LIN {X 0,Y 573.256,Z 464.198,A -85,B 0,C 180,E1 -2012.645,E2 -2012.645} C_VEL
LIN {X 0,Y 573.257,Z 464.201,A -85,B 0,C 180,E1 -2015.184,E2 -2015.184} C_VEL
LIN {X 0,Y 573.236,Z 464.206,A -85,B 0,C 180,E1 -2017.808,E2 -2017.808} C_VEL
LIN {X 0,Y 573.247,Z 464.198,A -85,B 0,C 180,E1 -2020.525,E2 -2020.525} C_VEL
LIN {X 0,Y 573.239,Z 464.205,A -85,B 0,C 180,E1 -2023.359,E2 -2023.359} C_VEL
LIN {X 0,Y 573.256,Z 464.197,A -85,B 0,C 180,E1 -2026.33,E2 -2026.33} C_VEL
LIN {X 0,Y 573.242,Z 464.198,A -85,B 0,C 180,E1 -2028.544,E2 -2028.544} C_VEL
LIN {X 0,Y 573.245,Z 464.204,A -85,B 0,C 180,E1 -2031.298,E2 -2031.298} C_VEL
LIN {X 0,Y 573.215,Z 464.205,A -85,B 0,C 180,E1 -2034.018,E2 -2034.018} C_VEL
LIN {X 0,Y 573.272,Z 464.195,A -85,B 0,C 180,E1 -2036.518,E2 -2036.518} C_VEL
LIN {X 0,Y 573.232,Z 464.203,A -85,B 0,C 180,E1 -2039.118,E2 -2039.118} C_VEL
LIN {X 0,Y 573.255,Z 464.2,A -85,B 0,C 180,E1 -2041.971,E2 -2041.971} C_VEL
LIN {X 0,Y 573.255,Z 464.197,A -85,B 0,C 180,E1 -2044.59,E2 -2044.59} C_VEL
LIN {X 0,Y 573.238,Z 464.207,A -85,B 0,C 180,E1 -2047.662,E2 -2047.662} C_VEL
LIN {X 0,Y 573.278,Z 464.194,A -85,B 0,C 180,E1 -2050.67,E2 -2050.67} C_VEL
LIN {X 0,Y 573.256,Z 464.205,A -85,B 0,C 180,E1 -2053.622,E2 -2053.622} C_VEL
LIN {X 0,Y 573.276,Z 464.199,A -85,B 0,C 180,E1 -2055.807,E2 -2055.807} C_VEL
LIN {X 0,Y 573.265,Z 464.196,A -85,B 0,C 180,E1 -2058.745,E2 -2058.745} C_VEL
LIN {X 0,Y 573.309,Z 464.199,A -85,B 0,C 180,E1 -2061.541,E2 -2061.541} C_VEL
LIN {X 0,Y 573.291,Z 464.192,A -85,B 0,C 180,E1 -2064.372,E2 -2064.372} C_VEL
LIN {X 0,Y 573.316,Z 464.193,A -85,B 0,C 180,E1 -2067.892,E2 -2067.892} C_VEL
LIN {X 0,Y 573.33,Z 464.188,A -85,B 0,C 180,E1 -2070.702,E2 -2070.702} C_VEL
LIN {X 0,Y 573.306,Z 464.192,A -85,B 0,C 180,E1 -2072.811,E2 -2072.811} C_VEL
LIN {X 0,Y 573.301,Z 464.198,A -85,B 0,C 180,E1 -2075.628,E2 -2075.628} C_VEL
LIN {X 0,Y 573.286,Z 464.193,A -85,B 0,C 180,E1 -2078.459,E2 -2078.459} C_VEL
LIN {X 0,Y 573.274,Z 464.203,A -85,B 0,C 180,E1 -2081.312,E2 -2081.312} C_VEL
LIN {X 0,Y 573.284,Z 464.193,A -85,B 0,C 180,E1 -2084.425,E2 -2084.425} C_VEL
LIN {X 0,Y 573.261,Z 464.202,A -85,B 0,C 180,E1 -2087.112,E2 -2087.112} C_VEL
LIN {X 0,Y 573.254,Z 464.198,A -85,B 0,C 180,E1 -2090.077,E2 -2090.077} C_VEL
LIN {X 0,Y 573.237,Z 464.205,A -85,B 0,C 180,E1 -2093.099,E2 -2093.099} C_VEL
LIN {X 0,Y 573.257,Z 464.207,A -85,B 0,C 180,E1 -2095.41,E2 -2095.41} C_VEL
LIN {X 0,Y 573.253,Z 464.198,A -85,B 0,C 180,E1 -2098.029,E2 -2098.029} C_VEL
LIN {X 0,Y 573.236,Z 464.202,A -85,B 0,C 180,E1 -2100.883,E2 -2100.883} C_VEL
LIN {X 0,Y 573.264,Z 464.203,A -85,B 0,C 180,E1 -2103.524,E2 -2103.524} C_VEL
LIN {X 0,Y 573.216,Z 464.202,A -85,B 0,C 180,E1 -2106.052,E2 -2106.052} C_VEL
LIN {X 0,Y 573.25,Z 464.199,A -85,B 0,C 180,E1 -2108.701,E2 -2108.701} C_VEL
LIN {X 0,Y 573.256,Z 464.202,A -85,B 0,C 180,E1 -2111.596,E2 -2111.596} C_VEL
LIN {X 0,Y 573.24,Z 464.199,A -85,B 0,C 180,E1 -2114.333,E2 -2114.333} C_VEL
LIN {X 0,Y 573.242,Z 464.208,A -85,B 0,C 180,E1 -2117.359,E2 -2117.359} C_VEL
LIN {X 0,Y 573.254,Z 464.198,A -85,B 0,C 180,E1 -2120.567,E2 -2120.567} C_VEL
LIN {X 0,Y 573.254,Z 464.204,A -85,B 0,C 180,E1 -2123.078,E2 -2123.078} C_VEL
LIN {X 0,Y 573.274,Z 464.198,A -85,B 0,C 180,E1 -2125.672,E2 -2125.672} C_VEL
LIN {X 0,Y 573.242,Z 464.199,A -85,B 0,C 180,E1 -2128.185,E2 -2128.185} C_VEL
LIN {X 0,Y 573.268,Z 464.197,A -85,B 0,C 180,E1 -2130.634,E2 -2130.634} C_VEL
LIN {X 0,Y 573.241,Z 464.207,A -85,B 0,C 180,E1 -2133.507,E2 -2133.507} C_VEL
LIN {X 0,Y 573.301,Z 464.323,A -85,B 0,C 180,E1 -2135.416,E2 -2135.416} C_VEL
LIN {X 0,Y 574.239,Z 469.528,A -85,B 0,C 180,E1 -2136.179,E2 -2136.179} C_VEL
LIN {X 0,Y 574.011,Z 490.489,A -85,B 0,C 180,E1 -2139.034,E2 -2139.034} C_VEL
LIN {X 0,Y 573.735,Z 512.558,A -85,B 0,C 180,E1 -2141.983,E2 -2141.983} C_VEL
LIN {X 0,Y 573.512,Z 533.38,A -85,B 0,C 180,E1 -2144.724,E2 -2144.724} C_VEL
LIN {X 0,Y 573.435,Z 544.763,A -85,B 0,C 180,E1 -2146.207,E2 -2146.207} C_VEL
LIN {X 0,Y 574.111,Z 551.018,A -85,B 0,C 180,E1 -2146.302,E2 -2146.302} C_VEL
LIN {X 0,Y 573.879,Z 653.245,A -85,B 0,C 180,E1 -2147.602,E2 -2147.602} C_VEL
LIN {X 0,Y 573.815,Z 666.002,A -85,B 0,C 180,E1 -2147.893,E2 -2147.893} C_VEL
LIN {X 0,Y 573.683,Z 679.691,A -85,B 0,C 180,E1 -2148.374,E2 -2148.374} C_VEL
LIN {X 0,Y 573.588,Z 690.234,A -85,B 0,C 180,E1 -2148.874,E2 -2148.874} C_VEL
LIN {X 0,Y 573.456,Z 700.709,A -85,B 0,C 180,E1 -2149.496,E2 -2149.496} C_VEL
LIN {X 0,Y 573.35,Z 711.515,A -85,B 0,C 180,E1 -2150.297,E2 -2150.297} C_VEL
LIN {X 0,Y 573.241,Z 721.15,A -85,B 0,C 180,E1 -2151.185,E2 -2151.185} C_VEL
LIN {X 0,Y 573.161,Z 729.049,A -85,B 0,C 180,E1 -2152.071,E2 -2152.071} C_VEL
LIN {X 0,Y 573.112,Z 735.624,A -85,B 0,C 180,E1 -2152.956,E2 -2152.956} C_VEL
LIN {X 0,Y 573.078,Z 742.083,A -85,B 0,C 180,E1 -2154.017,E2 -2154.017} C_VEL
LIN {X 0,Y 572.962,Z 747.233,A -85,B 0,C 180,E1 -2155.074,E2 -2155.074} C_VEL
LIN {X 0,Y 573.015,Z 751.228,A -85,B 0,C 180,E1 -2156.132,E2 -2156.132} C_VEL
LIN {X 0,Y 572.959,Z 754.184,A -85,B 0,C 180,E1 -2157.188,E2 -2157.188} C_VEL
LIN {X 0,Y 572.947,Z 756.639,A -85,B 0,C 180,E1 -2158.594,E2 -2158.594} C_VEL
LIN {X 0,Y 572.941,Z 757.253,A -85,B 0,C 180,E1 -2159.297,E2 -2159.297} C_VEL
LIN {X 0,Y 572.941,Z 757.312,A -85,B 0,C 180,E1 -2160.703,E2 -2160.703} C_VEL
LIN {X 0,Y 572.946,Z 756.739,A -85,B 0,C 180,E1 -2161.406,E2 -2161.406} C_VEL
LIN {X 0,Y 572.96,Z 754.408,A -85,B 0,C 180,E1 -2162.812,E2 -2162.812} C_VEL
LIN {X 0,Y 573.014,Z 751.537,A -85,B 0,C 180,E1 -2163.868,E2 -2163.868} C_VEL
LIN {X 0,Y 572.963,Z 747.634,A -85,B 0,C 180,E1 -2164.926,E2 -2164.926} C_VEL
LIN {X 0,Y 573.073,Z 742.582,A -85,B 0,C 180,E1 -2165.983,E2 -2165.983} C_VEL
LIN {X 0,Y 573.082,Z 736.228,A -85,B 0,C 180,E1 -2167.044,E2 -2167.044} C_VEL
LIN {X 0,Y 573.175,Z 728.352,A -85,B 0,C 180,E1 -2168.106,E2 -2168.106} C_VEL
LIN {X 0,Y 573.287,Z 718.508,A -85,B 0,C 180,E1 -2169.17,E2 -2169.17} C_VEL
LIN {X 0,Y 573.409,Z 708.142,A -85,B 0,C 180,E1 -2170.059,E2 -2170.059} C_VEL
LIN {X 0,Y 573.512,Z 697.959,A -85,B 0,C 180,E1 -2170.769,E2 -2170.769} C_VEL
LIN {X 0,Y 573.654,Z 685.746,A -85,B 0,C 180,E1 -2171.447,E2 -2171.447} C_VEL
LIN {X 0,Y 573.723,Z 674.21,A -85,B 0,C 180,E1 -2171.93,E2 -2171.93} C_VEL
LIN {X 0,Y 573.848,Z 661.681,A -85,B 0,C 180,E1 -2172.309,E2 -2172.309} C_VEL
LIN {X 0,Y 573.91,Z 649.104,A -85,B 0,C 180,E1 -2172.554,E2 -2172.554} C_VEL
LIN {X 0,Y 573.973,Z 548.434,A -85,B 0,C 180,E1 -2173.824,E2 -2173.824} C_VEL
LIN {X 0,Y 573.446,Z 544.656,A -85,B 0,C 180,E1 -2173.895,E2 -2173.895} C_VEL
LIN {X 0,Y 573.672,Z 520.179,A -85,B 0,C 180,E1 -2177.099,E2 -2177.099} C_VEL
LIN {X 0,Y 573.909,Z 497.958,A -85,B 0,C 180,E1 -2180.053,E2 -2180.053} C_VEL
LIN {X 0,Y 574.222,Z 475.736,A -85,B 0,C 180,E1 -2183.057,E2 -2183.057} C_VEL
LIN {X 0,Y 574.216,Z 468.791,A -85,B 0,C 180,E1 -2184.014,E2 -2184.014} C_VEL
LIN {X 0,Y 573.301,Z 464.202,A -85,B 0,C 180,E1 -2184.718,E2 -2184.718} C_VEL
LIN {X 0,Y 573.269,Z 464.197,A -85,B 0,C 180,E1 -2187.766,E2 -2187.766} C_VEL
LIN {X 0,Y 573.249,Z 464.201,A -85,B 0,C 180,E1 -2190.176,E2 -2190.176} C_VEL
LIN {X 0,Y 573.256,Z 464.207,A -85,B 0,C 180,E1 -2192.645,E2 -2192.645} C_VEL
LIN {X 0,Y 573.212,Z 464.206,A -85,B 0,C 180,E1 -2195.188,E2 -2195.188} C_VEL
LIN {X 0,Y 573.237,Z 464.2,A -85,B 0,C 180,E1 -2197.808,E2 -2197.808} C_VEL
LIN {X 0,Y 573.247,Z 464.207,A -85,B 0,C 180,E1 -2200.525,E2 -2200.525} C_VEL
LIN {X 0,Y 573.238,Z 464.2,A -85,B 0,C 180,E1 -2203.359,E2 -2203.359} C_VEL
LIN {X 0,Y 573.256,Z 464.204,A -85,B 0,C 180,E1 -2206.33,E2 -2206.33} C_VEL
LIN {X 0,Y 573.248,Z 464.207,A -85,B 0,C 180,E1 -2208.544,E2 -2208.544} C_VEL
LIN {X 0,Y 573.245,Z 464.199,A -85,B 0,C 180,E1 -2211.298,E2 -2211.298} C_VEL
LIN {X 0,Y 573.262,Z 464.201,A -85,B 0,C 180,E1 -2214.012,E2 -2214.012} C_VEL
LIN {X 0,Y 573.288,Z 464.201,A -85,B 0,C 180,E1 -2216.519,E2 -2216.519} C_VEL
LIN {X 0,Y 573.246,Z 464.2,A -85,B 0,C 180,E1 -2219.115,E2 -2219.115} C_VEL
LIN {X 0,Y 573.255,Z 464.203,A -85,B 0,C 180,E1 -2221.971,E2 -2221.971} C_VEL
LIN {X 0,Y 573.259,Z 464.205,A -85,B 0,C 180,E1 -2224.59,E2 -2224.59} C_VEL
LIN {X 0,Y 573.278,Z 464.334,A -85,B 0,C 180,E1 -2226.259,E2 -2226.259} C_VEL
LIN {X 0,Y 574.399,Z 469.715,A -85,B 0,C 180,E1 -2226.95,E2 -2226.95} C_VEL
LIN {X 0,Y 574.101,Z 492.105,A -85,B 0,C 180,E1 -2229.581,E2 -2229.581} C_VEL
LIN {X 0,Y 573.84,Z 516.255,A -85,B 0,C 180,E1 -2232.373,E2 -2232.373} C_VEL
LIN {X 0,Y 573.76,Z 523.691,A -85,B 0,C 180,E1 -2233.225,E2 -2233.225} C_VEL
LIN {X 0,Y 574.613,Z 530.399,A -85,B 0,C 180,E1 -2233.342,E2 -2233.342} C_VEL
LIN {X 0,Y 574.277,Z 662.882,A -85,B 0,C 180,E1 -2235.04,E2 -2235.04} C_VEL
LIN {X 0,Y 574.174,Z 676.909,A -85,B 0,C 180,E1 -2235.363,E2 -2235.363} C_VEL
LIN {X 0,Y 574.005,Z 690.71,A -85,B 0,C 180,E1 -2235.825,E2 -2235.825} C_VEL
LIN {X 0,Y 573.869,Z 704.641,A -85,B 0,C 180,E1 -2236.454,E2 -2236.454} C_VEL
LIN {X 0,Y 573.711,Z 717.099,A -85,B 0,C 180,E1 -2237.172,E2 -2237.172} C_VEL
LIN {X 0,Y 573.533,Z 729.641,A -85,B 0,C 180,E1 -2238.066,E2 -2238.066} C_VEL
LIN {X 0,Y 573.437,Z 741.178,A -85,B 0,C 180,E1 -2239.084,E2 -2239.084} C_VEL
LIN {X 0,Y 573.239,Z 750.851,A -85,B 0,C 180,E1 -2240.117,E2 -2240.117} C_VEL
LIN {X 0,Y 573.202,Z 759.172,A -85,B 0,C 180,E1 -2241.184,E2 -2241.184} C_VEL
LIN {X 0,Y 573.11,Z 767.127,A -85,B 0,C 180,E1 -2242.425,E2 -2242.425} C_VEL
LIN {X 0,Y 573.02,Z 773.527,A -85,B 0,C 180,E1 -2243.663,E2 -2243.663} C_VEL
LIN {X 0,Y 573.001,Z 777.961,A -85,B 0,C 180,E1 -2244.722,E2 -2244.722} C_VEL
LIN {X 0,Y 573.028,Z 781.443,A -85,B 0,C 180,E1 -2245.78,E2 -2245.78} C_VEL
LIN {X 0,Y 572.956,Z 784.832,A -85,B 0,C 180,E1 -2247.188,E2 -2247.188} C_VEL
LIN {X 0,Y 572.941,Z 786.832,A -85,B 0,C 180,E1 -2248.594,E2 -2248.594} C_VEL
LIN {X 0,Y 572.937,Z 787.5,A -85,B 0,C 180,E1 -2250,E2 -2250} C_VEL
LIN {X 0,Y 572.941,Z 786.833,A -85,B 0,C 180,E1 -2251.406,E2 -2251.406} C_VEL
LIN {X 0,Y 572.956,Z 784.833,A -85,B 0,C 180,E1 -2252.812,E2 -2252.812} C_VEL
LIN {X 0,Y 573.028,Z 781.444,A -85,B 0,C 180,E1 -2254.22,E2 -2254.22} C_VEL
LIN {X 0,Y 573.059,Z 776.568,A -85,B 0,C 180,E1 -2255.631,E2 -2255.631} C_VEL
LIN {X 0,Y 573.058,Z 771.852,A -85,B 0,C 180,E1 -2256.693,E2 -2256.693} C_VEL
LIN {X 0,Y 573.126,Z 765.037,A -85,B 0,C 180,E1 -2257.93,E2 -2257.93} C_VEL
LIN {X 0,Y 573.225,Z 756.558,A -85,B 0,C 180,E1 -2259.171,E2 -2259.171} C_VEL
LIN {X 0,Y 573.304,Z 747.706,A -85,B 0,C 180,E1 -2260.239,E2 -2260.239} C_VEL
LIN {X 0,Y 573.462,Z 736.99,A -85,B 0,C 180,E1 -2261.308,E2 -2261.308} C_VEL
LIN {X 0,Y 573.616,Z 726.141,A -85,B 0,C 180,E1 -2262.201,E2 -2262.201} C_VEL
LIN {X 0,Y 573.739,Z 714.257,A -85,B 0,C 180,E1 -2263.008,E2 -2263.008} C_VEL
LIN {X 0,Y 573.956,Z 701.092,A -85,B 0,C 180,E1 -2263.724,E2 -2263.724} C_VEL
LIN {X 0,Y 574.077,Z 687.827,A -85,B 0,C 180,E1 -2264.284,E2 -2264.284} C_VEL
LIN {X 0,Y 574.2,Z 673.826,A -85,B 0,C 180,E1 -2264.72,E2 -2264.72} C_VEL
LIN {X 0,Y 574.308,Z 660.122,A -85,B 0,C 180,E1 -2265.005,E2 -2265.005} C_VEL
LIN {X 0,Y 574.555,Z 528.602,A -85,B 0,C 180,E1 -2266.683,E2 -2266.683} C_VEL
LIN {X 0,Y 573.762,Z 523.691,A -85,B 0,C 180,E1 -2266.775,E2 -2266.775} C_VEL
LIN {X 0,Y 574.03,Z 498.31,A -85,B 0,C 180,E1 -2269.698,E2 -2269.698} C_VEL
LIN {X 0,Y 574.393,Z 472.912,A -85,B 0,C 180,E1 -2272.67,E2 -2272.67} C_VEL
LIN {X 0,Y 574.251,Z 468.74,A -85,B 0,C 180,E1 -2273.172,E2 -2273.172} C_VEL
LIN {X 0,Y 573.26,Z 464.208,A -85,B 0,C 180,E1 -2273.783,E2 -2273.783} C_VEL
LIN {X 0,Y 573.241,Z 464.202,A -85,B 0,C 180,E1 -2276.493,E2 -2276.493} C_VEL
LIN {X 0,Y 573.241,Z 464.201,A -85,B 0,C 180,E1 -2278.564,E2 -2278.564} C_VEL
LIN {X 0,Y 573.239,Z 464.204,A -85,B 0,C 180,E1 -2280.993,E2 -2280.993} C_VEL
LIN {X 0,Y 573.265,Z 464.206,A -85,B 0,C 180,E1 -2283.524,E2 -2283.524} C_VEL
LIN {X 0,Y 573.216,Z 464.205,A -85,B 0,C 180,E1 -2286.052,E2 -2286.052} C_VEL
LIN {X 0,Y 573.245,Z 464.201,A -85,B 0,C 180,E1 -2288.702,E2 -2288.702} C_VEL
LIN {X 0,Y 573.24,Z 464.204,A -85,B 0,C 180,E1 -2291.594,E2 -2291.594} C_VEL
LIN {X 0,Y 573.241,Z 464.2,A -85,B 0,C 180,E1 -2294.333,E2 -2294.333} C_VEL
LIN {X 0,Y 573.243,Z 464.205,A -85,B 0,C 180,E1 -2297.359,E2 -2297.359} C_VEL
LIN {X 0,Y 573.252,Z 464.201,A -85,B 0,C 180,E1 -2300.393,E2 -2300.393} C_VEL
LIN {X 0,Y 573.256,Z 464.205,A -85,B 0,C 180,E1 -2303.078,E2 -2303.078} C_VEL
LIN {X 0,Y 573.275,Z 464.196,A -85,B 0,C 180,E1 -2305.672,E2 -2305.672} C_VEL
LIN {X 0,Y 573.252,Z 464.201,A -85,B 0,C 180,E1 -2308.185,E2 -2308.185} C_VEL
LIN {X 0,Y 573.269,Z 464.206,A -85,B 0,C 180,E1 -2310.634,E2 -2310.634} C_VEL
LIN {X 0,Y 573.242,Z 464.203,A -85,B 0,C 180,E1 -2313.507,E2 -2313.507} C_VEL
LIN {X 0,Y 573.235,Z 464.207,A -85,B 0,C 180,E1 -2316.135,E2 -2316.135} C_VEL
LIN {X 0,Y 573.279,Z 464.324,A -85,B 0,C 180,E1 -2316.652,E2 -2316.652} C_VEL
LIN {X 0,Y 574.225,Z 470.158,A -85,B 0,C 180,E1 -2317.513,E2 -2317.513} C_VEL
LIN {X 0,Y 573.938,Z 490.488,A -85,B 0,C 180,E1 -2320.316,E2 -2320.316} C_VEL
LIN {X 0,Y 573.712,Z 512.272,A -85,B 0,C 180,E1 -2323.269,E2 -2323.269} C_VEL
LIN {X 0,Y 573.495,Z 534.041,A -85,B 0,C 180,E1 -2326.174,E2 -2326.174} C_VEL
LIN {X 0,Y 573.41,Z 542.034,A -85,B 0,C 180,E1 -2327.21,E2 -2327.21} C_VEL
LIN {X 0,Y 574.076,Z 547.275,A -85,B 0,C 180,E1 -2327.292,E2 -2327.292} C_VEL
LIN {X 0,Y 573.864,Z 651.442,A -85,B 0,C 180,E1 -2328.62,E2 -2328.62} C_VEL
LIN {X 0,Y 573.79,Z 664.697,A -85,B 0,C 180,E1 -2328.944,E2 -2328.944} C_VEL
LIN {X 0,Y 573.632,Z 677.585,A -85,B 0,C 180,E1 -2329.41,E2 -2329.41} C_VEL
LIN {X 0,Y 573.551,Z 690.172,A -85,B 0,C 180,E1 -2330.033,E2 -2330.033} C_VEL
LIN {X 0,Y 573.429,Z 701.33,A -85,B 0,C 180,E1 -2330.743,E2 -2330.743} C_VEL
LIN {X 0,Y 573.358,Z 711.367,A -85,B 0,C 180,E1 -2331.542,E2 -2331.542} C_VEL
LIN {X 0,Y 573.22,Z 720.453,A -85,B 0,C 180,E1 -2332.426,E2 -2332.426} C_VEL
LIN {X 0,Y 573.147,Z 728.15,A -85,B 0,C 180,E1 -2333.333,E2 -2333.333} C_VEL
LIN {X 0,Y 573.087,Z 735.324,A -85,B 0,C 180,E1 -2334.37,E2 -2334.37} C_VEL
LIN {X 0,Y 573.049,Z 741.257,A -85,B 0,C 180,E1 -2335.428,E2 -2335.428} C_VEL
LIN {X 0,Y 573.057,Z 745.914,A -85,B 0,C 180,E1 -2336.484,E2 -2336.484} C_VEL
LIN {X 0,Y 573.016,Z 749.499,A -85,B 0,C 180,E1 -2337.54,E2 -2337.54} C_VEL
LIN {X 0,Y 572.949,Z 752.06,A -85,B 0,C 180,E1 -2338.594,E2 -2338.594} C_VEL
LIN {X 0,Y 572.941,Z 753.255,A -85,B 0,C 180,E1 -2339.297,E2 -2339.297} C_VEL
LIN {X 0,Y 572.939,Z 754.046,A -85,B 0,C 180,E1 -2340,E2 -2340} C_VEL
LIN {X 0,Y 572.946,Z 754.423,A -85,B 0,C 180,E1 -2341.406,E2 -2341.406} C_VEL
LIN {X 0,Y 572.936,Z 754.029,A -85,B 0,C 180,E1 -2342.109,E2 -2342.109} C_VEL
LIN {X 0,Y 572.955,Z 753.224,A -85,B 0,C 180,E1 -2342.812,E2 -2342.812} C_VEL
LIN {X 0,Y 573.009,Z 752.016,A -85,B 0,C 180,E1 -2343.516,E2 -2343.516} C_VEL
LIN {X 0,Y 573.005,Z 749.431,A -85,B 0,C 180,E1 -2344.573,E2 -2344.573} C_VEL
LIN {X 0,Y 573.051,Z 745.811,A -85,B 0,C 180,E1 -2345.631,E2 -2345.631} C_VEL
LIN {X 0,Y 573.045,Z 740.614,A -85,B 0,C 180,E1 -2346.788,E2 -2346.788} C_VEL
LIN {X 0,Y 573.112,Z 734.002,A -85,B 0,C 180,E1 -2347.93,E2 -2347.93} C_VEL
LIN {X 0,Y 573.173,Z 726.271,A -85,B 0,C 180,E1 -2348.994,E2 -2348.994} C_VEL
LIN {X 0,Y 573.226,Z 718.386,A -85,B 0,C 180,E1 -2349.884,E2 -2349.884} C_VEL
LIN {X 0,Y 573.374,Z 708.992,A -85,B 0,C 180,E1 -2350.752,E2 -2350.752} C_VEL
LIN {X 0,Y 573.454,Z 697.98,A -85,B 0,C 180,E1 -2351.577,E2 -2351.577} C_VEL
LIN {X 0,Y 573.62,Z 687.553,A -85,B 0,C 180,E1 -2352.201,E2 -2352.201} C_VEL
LIN {X 0,Y 573.683,Z 676.198,A -85,B 0,C 180,E1 -2352.739,E2 -2352.739} C_VEL
LIN {X 0,Y 573.777,Z 663.293,A -85,B 0,C 180,E1 -2353.187,E2 -2353.187} C_VEL
LIN {X 0,Y 573.861,Z 651.004,A -85,B 0,C 180,E1 -2353.478,E2 -2353.478} C_VEL
LIN {X 0,Y 574.047,Z 583.153,A -85,B 0,C 180,E1 -2354.346,E2 -2354.346} C_VEL
LIN {X 0,Y 573.412,Z 577.345,A -85,B 0,C 180,E1 -2354.435,E2 -2354.435} C_VEL
LIN {X 0,Y 567.826,Z 558.666,A -85,B 0,C 180,E1 -2354.807,E2 -2354.807} C_VEL
LIN {X 0,Y 567.175,Z 552.859,A -85,B 0,C 180,E1 -2354.897,E2 -2354.897} C_VEL
LIN {X 0,Y 566.989,Z 545.666,A -85,B 0,C 180,E1 -2354.994,E2 -2354.994} C_VEL
LIN {X 0,Y 566.414,Z 541.802,A -85,B 0,C 180,E1 -2355.064,E2 -2355.064} C_VEL
LIN {X 0,Y 566.686,Z 519.515,A -85,B 0,C 180,E1 -2358.062,E2 -2358.062} C_VEL
LIN {X 0,Y 566.908,Z 498.879,A -85,B 0,C 180,E1 -2360.88,E2 -2360.88} C_VEL
LIN {X 0,Y 567.218,Z 479.798,A -85,B 0,C 180,E1 -2363.525,E2 -2363.525} C_VEL
LIN {X 0,Y 567.204,Z 469.946,A -85,B 0,C 180,E1 -2364.915,E2 -2364.915} C_VEL
LIN {X 0,Y 566.23,Z 465.076,A -85,B 0,C 180,E1 -2365.664,E2 -2365.664} C_VEL
LIN {X 0,Y 566.207,Z 465.079,A -85,B 0,C 180,E1 -2368.202,E2 -2368.202} C_VEL
LIN {X 0,Y 566.193,Z 465.08,A -85,B 0,C 180,E1 -2371.076,E2 -2371.076} C_VEL
LIN {X 0,Y 566.216,Z 465.083,A -85,B 0,C 180,E1 -2373.734,E2 -2373.734} C_VEL
LIN {X 0,Y 566.209,Z 465.075,A -85,B 0,C 180,E1 -2376.569,E2 -2376.569} C_VEL
LIN {X 0,Y 566.223,Z 465.082,A -85,B 0,C 180,E1 -2379.686,E2 -2379.686} C_VEL
LIN {X 0,Y 566.203,Z 465.076,A -85,B 0,C 180,E1 -2382.917,E2 -2382.917} C_VEL
LIN {X 0,Y 566.205,Z 465.078,A -85,B 0,C 180,E1 -2386.048,E2 -2386.048} C_VEL
LIN {X 0,Y 566.182,Z 465.079,A -85,B 0,C 180,E1 -2388.861,E2 -2388.861} C_VEL
LIN {X 0,Y 566.189,Z 465.086,A -85,B 0,C 180,E1 -2391.637,E2 -2391.637} C_VEL
LIN {X 0,Y 566.164,Z 465.081,A -85,B 0,C 180,E1 -2394.308,E2 -2394.308} C_VEL
LIN {X 0,Y 566.223,Z 465.074,A -85,B 0,C 180,E1 -2396.898,E2 -2396.898} C_VEL
LIN {X 0,Y 566.184,Z 465.086,A -85,B 0,C 180,E1 -2399.407,E2 -2399.407} C_VEL
LIN {X 0,Y 566.214,Z 465.079,A -85,B 0,C 180,E1 -2401.857,E2 -2401.857} C_VEL
LIN {X 0,Y 566.215,Z 465.075,A -85,B 0,C 180,E1 -2404.251,E2 -2404.251} C_VEL
LIN {X 0,Y 566.172,Z 465.08,A -85,B 0,C 180,E1 -2406.719,E2 -2406.719} C_VEL
LIN {X 0,Y 566.217,Z 465.081,A -85,B 0,C 180,E1 -2409.663,E2 -2409.663} C_VEL
LIN {X 0,Y 566.203,Z 465.076,A -85,B 0,C 180,E1 -2412.668,E2 -2412.668} C_VEL
LIN {X 0,Y 566.237,Z 465.079,A -85,B 0,C 180,E1 -2415.627,E2 -2415.627} C_VEL
LIN {X 0,Y 566.237,Z 465.071,A -85,B 0,C 180,E1 -2418.675,E2 -2418.675} C_VEL
LIN {X 0,Y 566.25,Z 465.079,A -85,B 0,C 180,E1 -2421.435,E2 -2421.435} C_VEL
LIN {X 0,Y 566.26,Z 465.069,A -85,B 0,C 180,E1 -2424.302,E2 -2424.302} C_VEL
LIN {X 0,Y 566.287,Z 465.069,A -85,B 0,C 180,E1 -2427.866,E2 -2427.866} C_VEL
LIN {X 0,Y 566.302,Z 465.064,A -85,B 0,C 180,E1 -2430.711,E2 -2430.711} C_VEL
LIN {X 0,Y 566.273,Z 465.068,A -85,B 0,C 180,E1 -2432.846,E2 -2432.846} C_VEL
LIN {X 0,Y 566.268,Z 465.073,A -85,B 0,C 180,E1 -2435.698,E2 -2435.698} C_VEL
LIN {X 0,Y 566.23,Z 465.072,A -85,B 0,C 180,E1 -2438.566,E2 -2438.566} C_VEL
LIN {X 0,Y 566.244,Z 465.08,A -85,B 0,C 180,E1 -2441.454,E2 -2441.454} C_VEL
LIN {X 0,Y 566.237,Z 465.071,A -85,B 0,C 180,E1 -2444.507,E2 -2444.507} C_VEL
LIN {X 0,Y 566.202,Z 465.085,A -85,B 0,C 180,E1 -2447.332,E2 -2447.332} C_VEL
LIN {X 0,Y 566.215,Z 465.074,A -85,B 0,C 180,E1 -2450.337,E2 -2450.337} C_VEL
LIN {X 0,Y 566.192,Z 465.087,A -85,B 0,C 180,E1 -2453.404,E2 -2453.404} C_VEL
LIN {X 0,Y 566.216,Z 465.078,A -85,B 0,C 180,E1 -2455.749,E2 -2455.749} C_VEL
LIN {X 0,Y 566.205,Z 465.075,A -85,B 0,C 180,E1 -2458.202,E2 -2458.202} C_VEL
LIN {X 0,Y 566.197,Z 465.082,A -85,B 0,C 180,E1 -2461.077,E2 -2461.077} C_VEL
LIN {X 0,Y 566.214,Z 465.078,A -85,B 0,C 180,E1 -2463.734,E2 -2463.734} C_VEL
LIN {X 0,Y 566.201,Z 465.076,A -85,B 0,C 180,E1 -2466.57,E2 -2466.57} C_VEL
LIN {X 0,Y 566.223,Z 465.082,A -85,B 0,C 180,E1 -2469.273,E2 -2469.273} C_VEL
LIN {X 0,Y 566.217,Z 465.074,A -85,B 0,C 180,E1 -2472.087,E2 -2472.087} C_VEL
LIN {X 0,Y 566.171,Z 465.085,A -85,B 0,C 180,E1 -2475.036,E2 -2475.036} C_VEL
LIN {X 0,Y 566.191,Z 465.078,A -85,B 0,C 180,E1 -2477.911,E2 -2477.911} C_VEL
LIN {X 0,Y 566.224,Z 465.075,A -85,B 0,C 180,E1 -2480.727,E2 -2480.727} C_VEL
LIN {X 0,Y 566.187,Z 465.08,A -85,B 0,C 180,E1 -2483.788,E2 -2483.788} C_VEL
LIN {X 0,Y 566.215,Z 465.074,A -85,B 0,C 180,E1 -2486.266,E2 -2486.266} C_VEL
LIN {X 0,Y 566.193,Z 465.082,A -85,B 0,C 180,E1 -2488.924,E2 -2488.924} C_VEL
LIN {X 0,Y 566.215,Z 465.076,A -85,B 0,C 180,E1 -2491.858,E2 -2491.858} C_VEL
LIN {X 0,Y 566.218,Z 465.077,A -85,B 0,C 180,E1 -2494.251,E2 -2494.251} C_VEL
LIN {X 0,Y 566.257,Z 465.139,A -85,B 0,C 180,E1 -2495.236,E2 -2495.236} C_VEL
LIN {X 0,Y 567.333,Z 470.814,A -85,B 0,C 180,E1 -2496.059,E2 -2496.059} C_VEL
LIN {X 0,Y 567.15,Z 487.375,A -85,B 0,C 180,E1 -2498.34,E2 -2498.34} C_VEL
LIN {X 0,Y 566.86,Z 508.398,A -85,B 0,C 180,E1 -2501.195,E2 -2501.195} C_VEL
LIN {X 0,Y 566.596,Z 529.22,A -85,B 0,C 180,E1 -2503.979,E2 -2503.979} C_VEL
LIN {X 0,Y 566.451,Z 544.806,A -85,B 0,C 180,E1 -2506.033,E2 -2506.033} C_VEL
LIN {X 0,Y 567.209,Z 551.063,A -85,B 0,C 180,E1 -2506.132,E2 -2506.132} C_VEL
LIN {X 0,Y 566.964,Z 653.236,A -85,B 0,C 180,E1 -2507.449,E2 -2507.449} C_VEL
LIN {X 0,Y 566.888,Z 665.22,A -85,B 0,C 180,E1 -2507.72,E2 -2507.72} C_VEL
LIN {X 0,Y 566.741,Z 678.551,A -85,B 0,C 180,E1 -2508.18,E2 -2508.18} C_VEL
LIN {X 0,Y 566.63,Z 689.626,A -85,B 0,C 180,E1 -2508.703,E2 -2508.703} C_VEL
LIN {X 0,Y 566.485,Z 699.317,A -85,B 0,C 180,E1 -2509.275,E2 -2509.275} C_VEL
LIN {X 0,Y 566.342,Z 709.296,A -85,B 0,C 180,E1 -2509.995,E2 -2509.995} C_VEL
LIN {X 0,Y 566.238,Z 719.401,A -85,B 0,C 180,E1 -2510.895,E2 -2510.895} C_VEL
LIN {X 0,Y 566.134,Z 727.61,A -85,B 0,C 180,E1 -2511.792,E2 -2511.792} C_VEL
LIN {X 0,Y 566.05,Z 735.619,A -85,B 0,C 180,E1 -2512.868,E2 -2512.868} C_VEL
LIN {X 0,Y 565.994,Z 742.079,A -85,B 0,C 180,E1 -2513.941,E2 -2513.941} C_VEL
LIN {X 0,Y 565.877,Z 747.229,A -85,B 0,C 180,E1 -2515.013,E2 -2515.013} C_VEL
LIN {X 0,Y 565.926,Z 751.226,A -85,B 0,C 180,E1 -2516.084,E2 -2516.084} C_VEL
LIN {X 0,Y 565.878,Z 754.183,A -85,B 0,C 180,E1 -2517.152,E2 -2517.152} C_VEL
LIN {X 0,Y 565.846,Z 756.64,A -85,B 0,C 180,E1 -2518.577,E2 -2518.577} C_VEL
LIN {X 0,Y 565.841,Z 757.253,A -85,B 0,C 180,E1 -2519.288,E2 -2519.288} C_VEL
LIN {X 0,Y 565.841,Z 757.311,A -85,B 0,C 180,E1 -2520.712,E2 -2520.712} C_VEL
LIN {X 0,Y 565.846,Z 756.74,A -85,B 0,C 180,E1 -2521.423,E2 -2521.423} C_VEL
LIN {X 0,Y 565.878,Z 754.404,A -85,B 0,C 180,E1 -2522.848,E2 -2522.848} C_VEL
LIN {X 0,Y 565.926,Z 751.533,A -85,B 0,C 180,E1 -2523.916,E2 -2523.916} C_VEL
LIN {X 0,Y 565.878,Z 747.627,A -85,B 0,C 180,E1 -2524.987,E2 -2524.987} C_VEL
LIN {X 0,Y 565.989,Z 742.571,A -85,B 0,C 180,E1 -2526.059,E2 -2526.059} C_VEL
LIN {X 0,Y 566.031,Z 736.215,A -85,B 0,C 180,E1 -2527.132,E2 -2527.132} C_VEL
LIN {X 0,Y 566.111,Z 729.754,A -85,B 0,C 180,E1 -2528.028,E2 -2528.028} C_VEL
LIN {X 0,Y 566.206,Z 721.988,A -85,B 0,C 180,E1 -2528.926,E2 -2528.926} C_VEL
LIN {X 0,Y 566.33,Z 712.582,A -85,B 0,C 180,E1 -2529.825,E2 -2529.825} C_VEL
LIN {X 0,Y 566.461,Z 702.075,A -85,B 0,C 180,E1 -2530.635,E2 -2530.635} C_VEL
LIN {X 0,Y 566.629,Z 691.48,A -85,B 0,C 180,E1 -2531.287,E2 -2531.287} C_VEL
LIN {X 0,Y 566.723,Z 680.914,A -85,B 0,C 180,E1 -2531.807,E2 -2531.807} C_VEL
LIN {X 0,Y 566.871,Z 668.942,A -85,B 0,C 180,E1 -2532.258,E2 -2532.258} C_VEL
LIN {X 0,Y 566.94,Z 654.517,A -85,B 0,C 180,E1 -2532.62,E2 -2532.62} C_VEL
LIN {X 0,Y 567.085,Z 613.565,A -85,B 0,C 180,E1 -2533.163,E2 -2533.163} C_VEL
LIN {X 0,Y 567.081,Z 549.159,A -85,B 0,C 180,E1 -2533.985,E2 -2533.985} C_VEL
LIN {X 0,Y 566.459,Z 544.652,A -85,B 0,C 180,E1 -2534.069,E2 -2534.069} C_VEL
LIN {X 0,Y 566.696,Z 521.526,A -85,B 0,C 180,E1 -2537.135,E2 -2537.135} C_VEL
LIN {X 0,Y 566.95,Z 500.734,A -85,B 0,C 180,E1 -2539.931,E2 -2539.931} C_VEL
LIN {X 0,Y 567.317,Z 478.509,A -85,B 0,C 180,E1 -2542.969,E2 -2542.969} C_VEL
LIN {X 0,Y 567.387,Z 471.235,A -85,B 0,C 180,E1 -2543.954,E2 -2543.954} C_VEL
LIN {X 0,Y 566.251,Z 465.08,A -85,B 0,C 180,E1 -2544.813,E2 -2544.813} C_VEL
LIN {X 0,Y 566.211,Z 465.079,A -85,B 0,C 180,E1 -2547.339,E2 -2547.339} C_VEL
LIN {X 0,Y 566.204,Z 465.077,A -85,B 0,C 180,E1 -2549.769,E2 -2549.769} C_VEL
LIN {X 0,Y 566.206,Z 465.083,A -85,B 0,C 180,E1 -2552.43,E2 -2552.43} C_VEL
LIN {X 0,Y 566.185,Z 465.084,A -85,B 0,C 180,E1 -2554.99,E2 -2554.99} C_VEL
LIN {X 0,Y 566.198,Z 465.077,A -85,B 0,C 180,E1 -2557.461,E2 -2557.461} C_VEL
LIN {X 0,Y 566.212,Z 465.079,A -85,B 0,C 180,E1 -2560.199,E2 -2560.199} C_VEL
LIN {X 0,Y 566.202,Z 465.079,A -85,B 0,C 180,E1 -2563.054,E2 -2563.054} C_VEL
LIN {X 0,Y 566.205,Z 465.078,A -85,B 0,C 180,E1 -2566.048,E2 -2566.048} C_VEL
LIN {X 0,Y 566.186,Z 465.082,A -85,B 0,C 180,E1 -2568.861,E2 -2568.861} C_VEL
LIN {X 0,Y 566.189,Z 465.078,A -85,B 0,C 180,E1 -2571.637,E2 -2571.637} C_VEL
LIN {X 0,Y 566.208,Z 465.084,A -85,B 0,C 180,E1 -2574.311,E2 -2574.311} C_VEL
LIN {X 0,Y 566.232,Z 465.075,A -85,B 0,C 180,E1 -2576.898,E2 -2576.898} C_VEL
LIN {X 0,Y 566.196,Z 465.078,A -85,B 0,C 180,E1 -2579.408,E2 -2579.408} C_VEL
LIN {X 0,Y 566.214,Z 465.079,A -85,B 0,C 180,E1 -2581.857,E2 -2581.857} C_VEL
LIN {X 0,Y 566.219,Z 465.084,A -85,B 0,C 180,E1 -2584.251,E2 -2584.251} C_VEL
LIN {X 0,Y 566.229,Z 465.118,A -85,B 0,C 180,E1 -2586.04,E2 -2586.04} C_VEL
LIN {X 0,Y 567.564,Z 471.314,A -85,B 0,C 180,E1 -2586.849,E2 -2586.849} C_VEL
LIN {X 0,Y 567.206,Z 493.704,A -85,B 0,C 180,E1 -2589.511,E2 -2589.511} C_VEL
LIN {X 0,Y 566.871,Z 518.014,A -85,B 0,C 180,E1 -2592.354,E2 -2592.354} C_VEL
LIN {X 0,Y 566.807,Z 523.709,A -85,B 0,C 180,E1 -2593.015,E2 -2593.015} C_VEL
LIN {X 0,Y 567.795,Z 530.146,A -85,B 0,C 180,E1 -2593.133,E2 -2593.133} C_VEL
LIN {X 0,Y 567.436,Z 662.882,A -85,B 0,C 180,E1 -2594.855,E2 -2594.855} C_VEL
LIN {X 0,Y 567.281,Z 677.027,A -85,B 0,C 180,E1 -2595.185,E2 -2595.185} C_VEL
LIN {X 0,Y 567.117,Z 690.709,A -85,B 0,C 180,E1 -2595.65,E2 -2595.65} C_VEL
LIN {X 0,Y 566.945,Z 704.643,A -85,B 0,C 180,E1 -2596.286,E2 -2596.286} C_VEL
LIN {X 0,Y 566.767,Z 717.1,A -85,B 0,C 180,E1 -2597.012,E2 -2597.012} C_VEL
LIN {X 0,Y 566.573,Z 729.641,A -85,B 0,C 180,E1 -2597.917,E2 -2597.917} C_VEL
LIN {X 0,Y 566.446,Z 740.318,A -85,B 0,C 180,E1 -2598.861,E2 -2598.861} C_VEL
LIN {X 0,Y 566.206,Z 750.851,A -85,B 0,C 180,E1 -2599.993,E2 -2599.993} C_VEL
LIN {X 0,Y 566.137,Z 759.172,A -85,B 0,C 180,E1 -2601.073,E2 -2601.073} C_VEL
LIN {X 0,Y 566.046,Z 767.127,A -85,B 0,C 180,E1 -2602.33,E2 -2602.33} C_VEL
LIN {X 0,Y 565.944,Z 773.528,A -85,B 0,C 180,E1 -2603.583,E2 -2603.583} C_VEL
LIN {X 0,Y 565.928,Z 777.961,A -85,B 0,C 180,E1 -2604.656,E2 -2604.656} C_VEL
LIN {X 0,Y 565.956,Z 781.443,A -85,B 0,C 180,E1 -2605.727,E2 -2605.727} C_VEL
LIN {X 0,Y 565.874,Z 784.832,A -85,B 0,C 180,E1 -2607.152,E2 -2607.152} C_VEL
LIN {X 0,Y 565.84,Z 786.833,A -85,B 0,C 180,E1 -2608.577,E2 -2608.577} C_VEL
LIN {X 0,Y 565.837,Z 787.5,A -85,B 0,C 180,E1 -2610,E2 -2610} C_VEL
LIN {X 0,Y 565.84,Z 786.833,A -85,B 0,C 180,E1 -2611.423,E2 -2611.423} C_VEL
LIN {X 0,Y 565.874,Z 784.833,A -85,B 0,C 180,E1 -2612.848,E2 -2612.848} C_VEL
LIN {X 0,Y 565.956,Z 781.445,A -85,B 0,C 180,E1 -2614.273,E2 -2614.273} C_VEL
LIN {X 0,Y 565.988,Z 776.568,A -85,B 0,C 180,E1 -2615.701,E2 -2615.701} C_VEL
LIN {X 0,Y 565.993,Z 772.044,A -85,B 0,C 180,E1 -2616.739,E2 -2616.739} C_VEL
LIN {X 0,Y 566.047,Z 765.036,A -85,B 0,C 180,E1 -2618.029,E2 -2618.029} C_VEL
LIN {X 0,Y 566.177,Z 756.557,A -85,B 0,C 180,E1 -2619.287,E2 -2619.287} C_VEL
LIN {X 0,Y 566.294,Z 747.706,A -85,B 0,C 180,E1 -2620.367,E2 -2620.367} C_VEL
LIN {X 0,Y 566.485,Z 736.989,A -85,B 0,C 180,E1 -2621.449,E2 -2621.449} C_VEL
LIN {X 0,Y 566.608,Z 726.14,A -85,B 0,C 180,E1 -2622.355,E2 -2622.355} C_VEL
LIN {X 0,Y 566.779,Z 714.255,A -85,B 0,C 180,E1 -2623.171,E2 -2623.171} C_VEL
LIN {X 0,Y 567.048,Z 701.093,A -85,B 0,C 180,E1 -2623.895,E2 -2623.895} C_VEL
LIN {X 0,Y 567.184,Z 688.051,A -85,B 0,C 180,E1 -2624.454,E2 -2624.454} C_VEL
LIN {X 0,Y 567.332,Z 673.629,A -85,B 0,C 180,E1 -2624.907,E2 -2624.907} C_VEL
LIN {X 0,Y 567.461,Z 660.121,A -85,B 0,C 180,E1 -2625.19,E2 -2625.19} C_VEL
LIN {X 0,Y 567.709,Z 529.106,A -85,B 0,C 180,E1 -2626.884,E2 -2626.884} C_VEL
LIN {X 0,Y 566.819,Z 523.64,A -85,B 0,C 180,E1 -2626.993,E2 -2626.993} C_VEL
LIN {X 0,Y 567.135,Z 498.505,A -85,B 0,C 180,E1 -2629.924,E2 -2629.924} C_VEL
LIN {X 0,Y 567.542,Z 474.512,A -85,B 0,C 180,E1 -2632.767,E2 -2632.767} C_VEL
LIN {X 0,Y 567.559,Z 471.313,A -85,B 0,C 180,E1 -2633.151,E2 -2633.151} C_VEL
LIN {X 0,Y 566.246,Z 465.081,A -85,B 0,C 180,E1 -2633.984,E2 -2633.984} C_VEL
LIN {X 0,Y 566.212,Z 465.078,A -85,B 0,C 180,E1 -2636.66,E2 -2636.66} C_VEL
LIN {X 0,Y 566.195,Z 465.081,A -85,B 0,C 180,E1 -2638.953,E2 -2638.953} C_VEL
LIN {X 0,Y 566.204,Z 465.086,A -85,B 0,C 180,E1 -2641.421,E2 -2641.421} C_VEL
LIN {X 0,Y 566.212,Z 465.079,A -85,B 0,C 180,E1 -2643.956,E2 -2643.956} C_VEL
LIN {X 0,Y 566.202,Z 465.078,A -85,B 0,C 180,E1 -2646.57,E2 -2646.57} C_VEL
LIN {X 0,Y 566.218,Z 465.079,A -85,B 0,C 180,E1 -2649.686,E2 -2649.686} C_VEL
LIN {X 0,Y 566.208,Z 465.081,A -85,B 0,C 180,E1 -2652.918,E2 -2652.918} C_VEL
LIN {X 0,Y 566.197,Z 465.078,A -85,B 0,C 180,E1 -2656.049,E2 -2656.049} C_VEL
LIN {X 0,Y 566.223,Z 465.081,A -85,B 0,C 180,E1 -2659.213,E2 -2659.213} C_VEL
LIN {X 0,Y 566.193,Z 465.079,A -85,B 0,C 180,E1 -2661.637,E2 -2661.637} C_VEL
LIN {X 0,Y 566.178,Z 465.083,A -85,B 0,C 180,E1 -2664.309,E2 -2664.309} C_VEL
LIN {X 0,Y 566.233,Z 465.081,A -85,B 0,C 180,E1 -2666.899,E2 -2666.899} C_VEL
LIN {X 0,Y 566.192,Z 465.08,A -85,B 0,C 180,E1 -2669.408,E2 -2669.408} C_VEL
LIN {X 0,Y 566.216,Z 465.079,A -85,B 0,C 180,E1 -2671.858,E2 -2671.858} C_VEL
LIN {X 0,Y 566.219,Z 465.083,A -85,B 0,C 180,E1 -2674.251,E2 -2674.251} C_VEL
LIN {X 0,Y 566.218,Z 465.118,A -85,B 0,C 180,E1 -2676.452,E2 -2676.452} C_VEL
LIN {X 0,Y 567.351,Z 471.602,A -85,B 0,C 180,E1 -2677.418,E2 -2677.418} C_VEL
LIN {X 0,Y 567.012,Z 492.125,A -85,B 0,C 180,E1 -2680.279,E2 -2680.279} C_VEL
LIN {X 0,Y 566.735,Z 513.856,A -85,B 0,C 180,E1 -2683.259,E2 -2683.259} C_VEL
LIN {X 0,Y 566.499,Z 535.504,A -85,B 0,C 180,E1 -2686.183,E2 -2686.183} C_VEL
LIN {X 0,Y 566.413,Z 541.802,A -85,B 0,C 180,E1 -2687.026,E2 -2687.026} C_VEL
LIN {X 0,Y 567.202,Z 548.322,A -85,B 0,C 180,E1 -2687.136,E2 -2687.136} C_VEL
LIN {X 0,Y 566.947,Z 651.05,A -85,B 0,C 180,E1 -2688.459,E2 -2688.459} C_VEL
LIN {X 0,Y 566.839,Z 664.384,A -85,B 0,C 180,E1 -2688.784,E2 -2688.784} C_VEL
LIN {X 0,Y 566.73,Z 676.841,A -85,B 0,C 180,E1 -2689.234,E2 -2689.234} C_VEL
LIN {X 0,Y 566.635,Z 688.841,A -85,B 0,C 180,E1 -2689.82,E2 -2689.82} C_VEL
LIN {X 0,Y 566.421,Z 700.248,A -85,B 0,C 180,E1 -2690.537,E2 -2690.537} C_VEL
LIN {X 0,Y 566.336,Z 710.485,A -85,B 0,C 180,E1 -2691.346,E2 -2691.346} C_VEL
LIN {X 0,Y 566.161,Z 720.571,A -85,B 0,C 180,E1 -2692.331,E2 -2692.331} C_VEL
LIN {X 0,Y 566.071,Z 728.893,A -85,B 0,C 180,E1 -2693.334,E2 -2693.334} C_VEL
LIN {X 0,Y 565.989,Z 736.515,A -85,B 0,C 180,E1 -2694.478,E2 -2694.478} C_VEL
LIN {X 0,Y 565.965,Z 742.992,A -85,B 0,C 180,E1 -2695.727,E2 -2695.727} C_VEL
LIN {X 0,Y 565.933,Z 747.264,A -85,B 0,C 180,E1 -2696.796,E2 -2696.796} C_VEL
LIN {X 0,Y 565.857,Z 750.497,A -85,B 0,C 180,E1 -2697.865,E2 -2697.865} C_VEL
LIN {X 0,Y 565.849,Z 752.086,A -85,B 0,C 180,E1 -2698.577,E2 -2698.577} C_VEL
LIN {X 0,Y 565.841,Z 753.272,A -85,B 0,C 180,E1 -2699.288,E2 -2699.288} C_VEL
LIN {X 0,Y 565.84,Z 754.054,A -85,B 0,C 180,E1 -2700,E2 -2700} C_VEL
LIN {X 0,Y 565.846,Z 754.417,A -85,B 0,C 180,E1 -2701.423,E2 -2701.423} C_VEL
LIN {X 0,Y 565.837,Z 754.014,A -85,B 0,C 180,E1 -2702.135,E2 -2702.135} C_VEL
LIN {X 0,Y 565.874,Z 753.202,A -85,B 0,C 180,E1 -2702.848,E2 -2702.848} C_VEL
LIN {X 0,Y 565.915,Z 751.989,A -85,B 0,C 180,E1 -2703.56,E2 -2703.56} C_VEL
LIN {X 0,Y 565.896,Z 749.394,A -85,B 0,C 180,E1 -2704.63,E2 -2704.63} C_VEL
LIN {X 0,Y 565.977,Z 745.757,A -85,B 0,C 180,E1 -2705.701,E2 -2705.701} C_VEL
LIN {X 0,Y 565.97,Z 740.233,A -85,B 0,C 180,E1 -2706.936,E2 -2706.936} C_VEL
LIN {X 0,Y 566.04,Z 733.918,A -85,B 0,C 180,E1 -2708.029,E2 -2708.029} C_VEL
LIN {X 0,Y 566.126,Z 726.161,A -85,B 0,C 180,E1 -2709.107,E2 -2709.107} C_VEL
LIN {X 0,Y 566.194,Z 718.254,A -85,B 0,C 180,E1 -2710.008,E2 -2710.008} C_VEL
LIN {X 0,Y 566.368,Z 709.029,A -85,B 0,C 180,E1 -2710.871,E2 -2710.871} C_VEL
LIN {X 0,Y 566.447,Z 699.089,A -85,B 0,C 180,E1 -2711.631,E2 -2711.631} C_VEL
LIN {X 0,Y 566.63,Z 687.289,A -85,B 0,C 180,E1 -2712.354,E2 -2712.354} C_VEL
LIN {X 0,Y 566.753,Z 675.879,A -85,B 0,C 180,E1 -2712.898,E2 -2712.898} C_VEL
LIN {X 0,Y 566.835,Z 662.828,A -85,B 0,C 180,E1 -2713.352,E2 -2713.352} C_VEL
LIN {X 0,Y 566.945,Z 650.185,A -85,B 0,C 180,E1 -2713.646,E2 -2713.646} C_VEL
LIN {X 0,Y 567.175,Z 552.859,A -85,B 0,C 180,E1 -2714.897,E2 -2714.897} C_VEL
LIN {X 0,Y 566.414,Z 548.993,A -85,B 0,C 180,E1 -2714.986,E2 -2714.986} C_VEL
LIN {X 0,Y 564.678,Z 545.559,A -85,B 0,C 180,E1 -2715.135,E2 -2715.135} C_VEL
LIN {X 0,Y 561.923,Z 541.563,A -85,B 0,C 180,E1 -2715.413,E2 -2715.413} C_VEL
LIN {X 0,Y 560.203,Z 538.816,A -85,B 0,C 180,E1 -2715.682,E2 -2715.682} C_VEL
LIN {X 0,Y 559.48,Z 536.223,A -85,B 0,C 180,E1 -2716,E2 -2716} C_VEL
LIN {X 0,Y 559.738,Z 516.66,A -85,B 0,C 180,E1 -2718.674,E2 -2718.674} C_VEL
LIN {X 0,Y 560.021,Z 497.397,A -85,B 0,C 180,E1 -2721.342,E2 -2721.342} C_VEL
LIN {X 0,Y 560.373,Z 478.381,A -85,B 0,C 180,E1 -2724.015,E2 -2724.015} C_VEL
LIN {X 0,Y 560.27,Z 471.203,A -85,B 0,C 180,E1 -2725.047,E2 -2725.047} C_VEL
LIN {X 0,Y 559.191,Z 465.954,A -85,B 0,C 180,E1 -2725.871,E2 -2725.871} C_VEL
LIN {X 0,Y 559.167,Z 465.955,A -85,B 0,C 180,E1 -2728.529,E2 -2728.529} C_VEL
LIN {X 0,Y 559.149,Z 465.96,A -85,B 0,C 180,E1 -2731.273,E2 -2731.273} C_VEL
LIN {X 0,Y 559.171,Z 465.957,A -85,B 0,C 180,E1 -2733.949,E2 -2733.949} C_VEL
LIN {X 0,Y 559.145,Z 465.957,A -85,B 0,C 180,E1 -2737.108,E2 -2737.108} C_VEL
LIN {X 0,Y 559.167,Z 465.956,A -85,B 0,C 180,E1 -2739.942,E2 -2739.942} C_VEL
LIN {X 0,Y 559.16,Z 465.953,A -85,B 0,C 180,E1 -2742.744,E2 -2742.744} C_VEL
LIN {X 0,Y 559.157,Z 465.96,A -85,B 0,C 180,E1 -2745.76,E2 -2745.76} C_VEL
LIN {X 0,Y 559.187,Z 465.95,A -85,B 0,C 180,E1 -2748.232,E2 -2748.232} C_VEL
LIN {X 0,Y 559.177,Z 465.955,A -85,B 0,C 180,E1 -2751.192,E2 -2751.192} C_VEL
LIN {X 0,Y 559.141,Z 465.961,A -85,B 0,C 180,E1 -2753.789,E2 -2753.789} C_VEL
LIN {X 0,Y 559.165,Z 465.952,A -85,B 0,C 180,E1 -2756.425,E2 -2756.425} C_VEL
LIN {X 0,Y 559.158,Z 465.955,A -85,B 0,C 180,E1 -2758.981,E2 -2758.981} C_VEL
LIN {X 0,Y 559.171,Z 465.96,A -85,B 0,C 180,E1 -2761.619,E2 -2761.619} C_VEL
LIN {X 0,Y 559.183,Z 465.954,A -85,B 0,C 180,E1 -2763.903,E2 -2763.903} C_VEL
LIN {X 0,Y 559.142,Z 465.955,A -85,B 0,C 180,E1 -2766.571,E2 -2766.571} C_VEL
LIN {X 0,Y 559.183,Z 465.958,A -85,B 0,C 180,E1 -2769.395,E2 -2769.395} C_VEL
LIN {X 0,Y 559.151,Z 465.961,A -85,B 0,C 180,E1 -2771.686,E2 -2771.686} C_VEL
LIN {X 0,Y 559.171,Z 465.954,A -85,B 0,C 180,E1 -2773.948,E2 -2773.948} C_VEL
LIN {X 0,Y 559.176,Z 465.952,A -85,B 0,C 180,E1 -2776.184,E2 -2776.184} C_VEL
LIN {X 0,Y 559.198,Z 465.952,A -85,B 0,C 180,E1 -2779.133,E2 -2779.133} C_VEL
LIN {X 0,Y 559.211,Z 465.948,A -85,B 0,C 180,E1 -2782.054,E2 -2782.054} C_VEL
LIN {X 0,Y 559.257,Z 465.943,A -85,B 0,C 180,E1 -2784.953,E2 -2784.953} C_VEL
LIN {X 0,Y 559.258,Z 465.944,A -85,B 0,C 180,E1 -2787.839,E2 -2787.839} C_VEL
LIN {X 0,Y 559.272,Z 465.939,A -85,B 0,C 180,E1 -2790.72,E2 -2790.72} C_VEL
LIN {X 0,Y 559.241,Z 465.945,A -85,B 0,C 180,E1 -2792.881,E2 -2792.881} C_VEL
LIN {X 0,Y 559.236,Z 465.948,A -85,B 0,C 180,E1 -2795.77,E2 -2795.77} C_VEL
LIN {X 0,Y 559.189,Z 465.95,A -85,B 0,C 180,E1 -2798.674,E2 -2798.674} C_VEL
LIN {X 0,Y 559.208,Z 465.954,A -85,B 0,C 180,E1 -2801.6,E2 -2801.6} C_VEL
LIN {X 0,Y 559.202,Z 465.948,A -85,B 0,C 180,E1 -2804.596,E2 -2804.596} C_VEL
LIN {X 0,Y 559.161,Z 465.96,A -85,B 0,C 180,E1 -2807.557,E2 -2807.557} C_VEL
LIN {X 0,Y 559.174,Z 465.954,A -85,B 0,C 180,E1 -2809.837,E2 -2809.837} C_VEL
LIN {X 0,Y 559.144,Z 465.955,A -85,B 0,C 180,E1 -2812.153,E2 -2812.153} C_VEL
LIN {X 0,Y 559.182,Z 465.957,A -85,B 0,C 180,E1 -2815.187,E2 -2815.187} C_VEL
LIN {X 0,Y 559.183,Z 465.954,A -85,B 0,C 180,E1 -2817.712,E2 -2817.712} C_VEL
LIN {X 0,Y 559.157,Z 465.953,A -85,B 0,C 180,E1 -2820.183,E2 -2820.183} C_VEL
LIN {X 0,Y 559.159,Z 465.954,A -85,B 0,C 180,E1 -2822.715,E2 -2822.715} C_VEL
LIN {X 0,Y 559.129,Z 465.967,A -85,B 0,C 180,E1 -2825.324,E2 -2825.324} C_VEL
LIN {X 0,Y 559.137,Z 465.957,A -85,B 0,C 180,E1 -2828.017,E2 -2828.017} C_VEL
LIN {X 0,Y 559.193,Z 465.954,A -85,B 0,C 180,E1 -2831.054,E2 -2831.054} C_VEL
LIN {X 0,Y 559.165,Z 465.956,A -85,B 0,C 180,E1 -2833.732,E2 -2833.732} C_VEL
LIN {X 0,Y 559.147,Z 465.957,A -85,B 0,C 180,E1 -2836.804,E2 -2836.804} C_VEL
LIN {X 0,Y 559.157,Z 465.961,A -85,B 0,C 180,E1 -2839.188,E2 -2839.188} C_VEL
LIN {X 0,Y 559.136,Z 465.957,A -85,B 0,C 180,E1 -2841.983,E2 -2841.983} C_VEL
LIN {X 0,Y 559.137,Z 465.958,A -85,B 0,C 180,E1 -2844.787,E2 -2844.787} C_VEL
LIN {X 0,Y 559.159,Z 465.962,A -85,B 0,C 180,E1 -2847.365,E2 -2847.365} C_VEL
LIN {X 0,Y 559.151,Z 465.954,A -85,B 0,C 180,E1 -2850.143,E2 -2850.143} C_VEL
LIN {X 0,Y 559.172,Z 465.959,A -85,B 0,C 180,E1 -2853.098,E2 -2853.098} C_VEL
LIN {X 0,Y 559.203,Z 465.985,A -85,B 0,C 180,E1 -2855.077,E2 -2855.077} C_VEL
LIN {X 0,Y 560.415,Z 472.089,A -85,B 0,C 180,E1 -2855.948,E2 -2855.948} C_VEL
LIN {X 0,Y 560.273,Z 486.142,A -85,B 0,C 180,E1 -2857.894,E2 -2857.894} C_VEL
LIN {X 0,Y 559.936,Z 507.183,A -85,B 0,C 180,E1 -2860.786,E2 -2860.786} C_VEL
LIN {X 0,Y 559.654,Z 527.837,A -85,B 0,C 180,E1 -2863.588,E2 -2863.588} C_VEL
LIN {X 0,Y 559.465,Z 544.853,A -85,B 0,C 180,E1 -2865.855,E2 -2865.855} C_VEL
LIN {X 0,Y 560.339,Z 551.109,A -85,B 0,C 180,E1 -2865.959,E2 -2865.959} C_VEL
LIN {X 0,Y 560.051,Z 653.227,A -85,B 0,C 180,E1 -2867.291,E2 -2867.291} C_VEL
LIN {X 0,Y 559.939,Z 665.219,A -85,B 0,C 180,E1 -2867.565,E2 -2867.565} C_VEL
LIN {X 0,Y 559.79,Z 678.549,A -85,B 0,C 180,E1 -2868.031,E2 -2868.031} C_VEL
LIN {X 0,Y 559.669,Z 689.375,A -85,B 0,C 180,E1 -2868.547,E2 -2868.547} C_VEL
LIN {X 0,Y 559.503,Z 699.315,A -85,B 0,C 180,E1 -2869.14,E2 -2869.14} C_VEL
LIN {X 0,Y 559.354,Z 709.298,A -85,B 0,C 180,E1 -2869.869,E2 -2869.869} C_VEL
LIN {X 0,Y 559.211,Z 719.408,A -85,B 0,C 180,E1 -2870.779,E2 -2870.779} C_VEL
LIN {X 0,Y 559.099,Z 727.615,A -85,B 0,C 180,E1 -2871.688,E2 -2871.688} C_VEL
LIN {X 0,Y 558.985,Z 735.614,A -85,B 0,C 180,E1 -2872.777,E2 -2872.777} C_VEL
LIN {X 0,Y 558.913,Z 742.074,A -85,B 0,C 180,E1 -2873.864,E2 -2873.864} C_VEL
LIN {X 0,Y 558.798,Z 747.225,A -85,B 0,C 180,E1 -2874.949,E2 -2874.949} C_VEL
LIN {X 0,Y 558.844,Z 751.223,A -85,B 0,C 180,E1 -2876.034,E2 -2876.034} C_VEL
LIN {X 0,Y 558.799,Z 754.182,A -85,B 0,C 180,E1 -2877.116,E2 -2877.116} C_VEL
LIN {X 0,Y 558.746,Z 756.642,A -85,B 0,C 180,E1 -2878.559,E2 -2878.559} C_VEL
LIN {X 0,Y 558.742,Z 757.254,A -85,B 0,C 180,E1 -2879.279,E2 -2879.279} C_VEL
LIN {X 0,Y 558.741,Z 757.311,A -85,B 0,C 180,E1 -2880.721,E2 -2880.721} C_VEL
LIN {X 0,Y 558.745,Z 756.739,A -85,B 0,C 180,E1 -2881.442,E2 -2881.442} C_VEL
LIN {X 0,Y 558.8,Z 754.4,A -85,B 0,C 180,E1 -2882.884,E2 -2882.884} C_VEL
LIN {X 0,Y 558.844,Z 751.528,A -85,B 0,C 180,E1 -2883.966,E2 -2883.966} C_VEL
LIN {X 0,Y 558.798,Z 747.618,A -85,B 0,C 180,E1 -2885.051,E2 -2885.051} C_VEL
LIN {X 0,Y 558.909,Z 742.56,A -85,B 0,C 180,E1 -2886.136,E2 -2886.136} C_VEL
LIN {X 0,Y 558.972,Z 736.202,A -85,B 0,C 180,E1 -2887.223,E2 -2887.223} C_VEL
LIN {X 0,Y 559.047,Z 729.74,A -85,B 0,C 180,E1 -2888.131,E2 -2888.131} C_VEL
LIN {X 0,Y 559.161,Z 721.972,A -85,B 0,C 180,E1 -2889.039,E2 -2889.039} C_VEL
LIN {X 0,Y 559.308,Z 712.575,A -85,B 0,C 180,E1 -2889.949,E2 -2889.949} C_VEL
LIN {X 0,Y 559.48,Z 702.063,A -85,B 0,C 180,E1 -2890.769,E2 -2890.769} C_VEL
LIN {X 0,Y 559.669,Z 691.018,A -85,B 0,C 180,E1 -2891.453,E2 -2891.453} C_VEL
LIN {X 0,Y 559.746,Z 679.853,A -85,B 0,C 180,E1 -2892.002,E2 -2892.002} C_VEL
LIN {X 0,Y 559.947,Z 666.749,A -85,B 0,C 180,E1 -2892.481,E2 -2892.481} C_VEL
LIN {X 0,Y 560.029,Z 654.439,A -85,B 0,C 180,E1 -2892.779,E2 -2892.779} C_VEL
LIN {X 0,Y 560.179,Z 617.097,A -85,B 0,C 180,E1 -2893.282,E2 -2893.282} C_VEL
LIN {X 0,Y 560.214,Z 550.009,A -85,B 0,C 180,E1 -2894.149,E2 -2894.149} C_VEL
LIN {X 0,Y 559.455,Z 544.734,A -85,B 0,C 180,E1 -2894.238,E2 -2894.238} C_VEL
LIN {X 0,Y 559.71,Z 521.277,A -85,B 0,C 180,E1 -2897.389,E2 -2897.389} C_VEL
LIN {X 0,Y 560.082,Z 499.338,A -85,B 0,C 180,E1 -2900.378,E2 -2900.378} C_VEL
LIN {X 0,Y 560.321,Z 482.311,A -85,B 0,C 180,E1 -2902.687,E2 -2902.687} C_VEL
LIN {X 0,Y 560.346,Z 471.974,A -85,B 0,C 180,E1 -2904.055,E2 -2904.055} C_VEL
LIN {X 0,Y 559.229,Z 465.954,A -85,B 0,C 180,E1 -2904.895,E2 -2904.895} C_VEL
LIN {X 0,Y 559.159,Z 465.956,A -85,B 0,C 180,E1 -2907.713,E2 -2907.713} C_VEL
LIN {X 0,Y 559.156,Z 465.957,A -85,B 0,C 180,E1 -2910.183,E2 -2910.183} C_VEL
LIN {X 0,Y 559.159,Z 465.964,A -85,B 0,C 180,E1 -2912.715,E2 -2912.715} C_VEL
LIN {X 0,Y 559.131,Z 465.959,A -85,B 0,C 180,E1 -2915.324,E2 -2915.324} C_VEL
LIN {X 0,Y 559.137,Z 465.958,A -85,B 0,C 180,E1 -2918.017,E2 -2918.017} C_VEL
LIN {X 0,Y 559.157,Z 465.96,A -85,B 0,C 180,E1 -2920.812,E2 -2920.812} C_VEL
LIN {X 0,Y 559.141,Z 465.956,A -85,B 0,C 180,E1 -2923.734,E2 -2923.734} C_VEL
LIN {X 0,Y 559.171,Z 465.957,A -85,B 0,C 180,E1 -2926.801,E2 -2926.801} C_VEL
LIN {X 0,Y 559.162,Z 465.954,A -85,B 0,C 180,E1 -2929.188,E2 -2929.188} C_VEL
LIN {X 0,Y 559.136,Z 465.96,A -85,B 0,C 180,E1 -2931.982,E2 -2931.982} C_VEL
LIN {X 0,Y 559.152,Z 465.959,A -85,B 0,C 180,E1 -2934.784,E2 -2934.784} C_VEL
LIN {X 0,Y 559.177,Z 465.952,A -85,B 0,C 180,E1 -2937.361,E2 -2937.361} C_VEL
LIN {X 0,Y 559.192,Z 465.957,A -85,B 0,C 180,E1 -2940.135,E2 -2940.135} C_VEL
LIN {X 0,Y 559.174,Z 465.954,A -85,B 0,C 180,E1 -2943.172,E2 -2943.172} C_VEL
LIN {X 0,Y 559.213,Z 466.143,A -85,B 0,C 180,E1 -2945.843,E2 -2945.843} C_VEL
LIN {X 0,Y 560.732,Z 473.038,A -85,B 0,C 180,E1 -2946.76,E2 -2946.76} C_VEL
LIN {X 0,Y 560.305,Z 495.304,A -85,B 0,C 180,E1 -2949.439,E2 -2949.439} C_VEL
LIN {X 0,Y 559.94,Z 519.293,A -85,B 0,C 180,E1 -2952.28,E2 -2952.28} C_VEL
LIN {X 0,Y 559.876,Z 523.719,A -85,B 0,C 180,E1 -2952.799,E2 -2952.799} C_VEL
LIN {X 0,Y 561.022,Z 531.84,A -85,B 0,C 180,E1 -2952.945,E2 -2952.945} C_VEL
LIN {X 0,Y 560.595,Z 662.882,A -85,B 0,C 180,E1 -2954.666,E2 -2954.666} C_VEL
LIN {X 0,Y 560.42,Z 677.398,A -85,B 0,C 180,E1 -2955.011,E2 -2955.011} C_VEL
LIN {X 0,Y 560.214,Z 691.837,A -85,B 0,C 180,E1 -2955.515,E2 -2955.515} C_VEL
LIN {X 0,Y 560.04,Z 704.641,A -85,B 0,C 180,E1 -2956.113,E2 -2956.113} C_VEL
LIN {X 0,Y 559.821,Z 717.102,A -85,B 0,C 180,E1 -2956.848,E2 -2956.848} C_VEL
LIN {X 0,Y 559.596,Z 729.643,A -85,B 0,C 180,E1 -2957.764,E2 -2957.764} C_VEL
LIN {X 0,Y 559.427,Z 740.739,A -85,B 0,C 180,E1 -2958.762,E2 -2958.762} C_VEL
LIN {X 0,Y 559.186,Z 750.852,A -85,B 0,C 180,E1 -2959.866,E2 -2959.866} C_VEL
LIN {X 0,Y 559.073,Z 759.173,A -85,B 0,C 180,E1 -2960.959,E2 -2960.959} C_VEL
LIN {X 0,Y 558.972,Z 767.127,A -85,B 0,C 180,E1 -2962.232,E2 -2962.232} C_VEL
LIN {X 0,Y 558.872,Z 773.528,A -85,B 0,C 180,E1 -2963.501,E2 -2963.501} C_VEL
LIN {X 0,Y 558.858,Z 777.961,A -85,B 0,C 180,E1 -2964.588,E2 -2964.588} C_VEL
LIN {X 0,Y 558.865,Z 781.443,A -85,B 0,C 180,E1 -2965.673,E2 -2965.673} C_VEL
LIN {X 0,Y 558.796,Z 784.832,A -85,B 0,C 180,E1 -2967.116,E2 -2967.116} C_VEL
LIN {X 0,Y 558.74,Z 786.833,A -85,B 0,C 180,E1 -2968.559,E2 -2968.559} C_VEL
LIN {X 0,Y 558.738,Z 787.5,A -85,B 0,C 180,E1 -2970,E2 -2970} C_VEL
LIN {X 0,Y 558.74,Z 786.834,A -85,B 0,C 180,E1 -2971.442,E2 -2971.442} C_VEL
LIN {X 0,Y 558.796,Z 784.834,A -85,B 0,C 180,E1 -2972.884,E2 -2972.884} C_VEL
LIN {X 0,Y 558.865,Z 781.445,A -85,B 0,C 180,E1 -2974.327,E2 -2974.327} C_VEL
LIN {X 0,Y 558.917,Z 776.568,A -85,B 0,C 180,E1 -2975.773,E2 -2975.773} C_VEL
LIN {X 0,Y 558.907,Z 770.053,A -85,B 0,C 180,E1 -2977.224,E2 -2977.224} C_VEL
LIN {X 0,Y 559.028,Z 762.801,A -85,B 0,C 180,E1 -2978.495,E2 -2978.495} C_VEL
LIN {X 0,Y 559.146,Z 753.821,A -85,B 0,C 180,E1 -2979.77,E2 -2979.77} C_VEL
LIN {X 0,Y 559.351,Z 744.391,A -85,B 0,C 180,E1 -2980.864,E2 -2980.864} C_VEL
LIN {X 0,Y 559.518,Z 733.95,A -85,B 0,C 180,E1 -2981.87,E2 -2981.87} C_VEL
LIN {X 0,Y 559.714,Z 722.433,A -85,B 0,C 180,E1 -2982.786,E2 -2982.786} C_VEL
LIN {X 0,Y 559.933,Z 709.641,A -85,B 0,C 180,E1 -2983.612,E2 -2983.612} C_VEL
LIN {X 0,Y 560.193,Z 697.149,A -85,B 0,C 180,E1 -2984.253,E2 -2984.253} C_VEL
LIN {X 0,Y 560.363,Z 683.269,A -85,B 0,C 180,E1 -2984.805,E2 -2984.805} C_VEL
LIN {X 0,Y 560.517,Z 669.559,A -85,B 0,C 180,E1 -2985.196,E2 -2985.196} C_VEL
LIN {X 0,Y 560.619,Z 655.591,A -85,B 0,C 180,E1 -2985.45,E2 -2985.45} C_VEL
LIN {X 0,Y 560.97,Z 530.352,A -85,B 0,C 180,E1 -2987.076,E2 -2987.076} C_VEL
LIN {X 0,Y 559.874,Z 523.703,A -85,B 0,C 180,E1 -2987.203,E2 -2987.203} C_VEL
LIN {X 0,Y 560.222,Z 500.101,A -85,B 0,C 180,E1 -2989.99,E2 -2989.99} C_VEL
LIN {X 0,Y 560.692,Z 476.111,A -85,B 0,C 180,E1 -2992.866,E2 -2992.866} C_VEL
LIN {X 0,Y 560.741,Z 473.049,A -85,B 0,C 180,E1 -2993.239,E2 -2993.239} C_VEL
LIN {X 0,Y 559.174,Z 465.959,A -85,B 0,C 180,E1 -2994.208,E2 -2994.208} C_VEL
LIN {X 0,Y 559.173,Z 465.956,A -85,B 0,C 180,E1 -2996.902,E2 -2996.902} C_VEL
LIN {X 0,Y 559.153,Z 465.962,A -85,B 0,C 180,E1 -2999.858,E2 -2999.858} C_VEL
LIN {X 0,Y 559.161,Z 465.955,A -85,B 0,C 180,E1 -3002.715,E2 -3002.715} C_VEL
LIN {X 0,Y 559.129,Z 465.966,A -85,B 0,C 180,E1 -3005.324,E2 -3005.324} C_VEL
LIN {X 0,Y 559.136,Z 465.959,A -85,B 0,C 180,E1 -3008.018,E2 -3008.018} C_VEL
LIN {X 0,Y 559.16,Z 465.958,A -85,B 0,C 180,E1 -3010.812,E2 -3010.812} C_VEL
LIN {X 0,Y 559.166,Z 465.955,A -85,B 0,C 180,E1 -3013.732,E2 -3013.732} C_VEL
LIN {X 0,Y 559.148,Z 465.961,A -85,B 0,C 180,E1 -3016.804,E2 -3016.804} C_VEL
LIN {X 0,Y 559.177,Z 465.959,A -85,B 0,C 180,E1 -3019.189,E2 -3019.189} C_VEL
LIN {X 0,Y 559.138,Z 465.958,A -85,B 0,C 180,E1 -3021.983,E2 -3021.983} C_VEL
LIN {X 0,Y 559.145,Z 465.965,A -85,B 0,C 180,E1 -3024.786,E2 -3024.786} C_VEL
LIN {X 0,Y 559.178,Z 465.954,A -85,B 0,C 180,E1 -3027.362,E2 -3027.362} C_VEL
LIN {X 0,Y 559.154,Z 465.959,A -85,B 0,C 180,E1 -3030.142,E2 -3030.142} C_VEL
LIN {X 0,Y 559.174,Z 465.96,A -85,B 0,C 180,E1 -3033.098,E2 -3033.098} C_VEL
LIN {X 0,Y 559.181,Z 465.959,A -85,B 0,C 180,E1 -3036.088,E2 -3036.088} C_VEL
LIN {X 0,Y 559.203,Z 466.163,A -85,B 0,C 180,E1 -3036.286,E2 -3036.286} C_VEL
LIN {X 0,Y 560.455,Z 472.986,A -85,B 0,C 180,E1 -3037.319,E2 -3037.319} C_VEL
LIN {X 0,Y 560.087,Z 493.451,A -85,B 0,C 180,E1 -3040.196,E2 -3040.196} C_VEL
LIN {X 0,Y 559.801,Z 514.116,A -85,B 0,C 180,E1 -3043.067,E2 -3043.067} C_VEL
LIN {X 0,Y 559.514,Z 535.607,A -85,B 0,C 180,E1 -3046.007,E2 -3046.007} C_VEL
LIN {X 0,Y 559.429,Z 541.839,A -85,B 0,C 180,E1 -3046.853,E2 -3046.853} C_VEL
LIN {X 0,Y 560.309,Z 549.373,A -85,B 0,C 180,E1 -3046.975,E2 -3046.975} C_VEL
LIN {X 0,Y 560.044,Z 650.261,A -85,B 0,C 180,E1 -3048.288,E2 -3048.288} C_VEL
LIN {X 0,Y 559.934,Z 663.284,A -85,B 0,C 180,E1 -3048.598,E2 -3048.598} C_VEL
LIN {X 0,Y 559.781,Z 676.099,A -85,B 0,C 180,E1 -3049.053,E2 -3049.053} C_VEL
LIN {X 0,Y 559.696,Z 687.439,A -85,B 0,C 180,E1 -3049.601,E2 -3049.601} C_VEL
LIN {X 0,Y 559.435,Z 699.132,A -85,B 0,C 180,E1 -3050.327,E2 -3050.327} C_VEL
LIN {X 0,Y 559.342,Z 709.603,A -85,B 0,C 180,E1 -3051.146,E2 -3051.146} C_VEL
LIN {X 0,Y 559.14,Z 719.065,A -85,B 0,C 180,E1 -3052.053,E2 -3052.053} C_VEL
LIN {X 0,Y 559.056,Z 726.926,A -85,B 0,C 180,E1 -3052.978,E2 -3052.978} C_VEL
LIN {X 0,Y 559.005,Z 734.368,A -85,B 0,C 180,E1 -3054.046,E2 -3054.046} C_VEL
LIN {X 0,Y 558.832,Z 739.566,A -85,B 0,C 180,E1 -3054.949,E2 -3054.949} C_VEL
LIN {X 0,Y 558.862,Z 744.588,A -85,B 0,C 180,E1 -3056.034,E2 -3056.034} C_VEL
LIN {X 0,Y 558.816,Z 748.507,A -85,B 0,C 180,E1 -3057.116,E2 -3057.116} C_VEL
LIN {X 0,Y 558.765,Z 750.531,A -85,B 0,C 180,E1 -3057.838,E2 -3057.838} C_VEL
LIN {X 0,Y 558.749,Z 752.113,A -85,B 0,C 180,E1 -3058.558,E2 -3058.558} C_VEL
LIN {X 0,Y 558.742,Z 753.288,A -85,B 0,C 180,E1 -3059.279,E2 -3059.279} C_VEL
LIN {X 0,Y 558.741,Z 754.062,A -85,B 0,C 180,E1 -3060,E2 -3060} C_VEL
LIN {X 0,Y 558.745,Z 754.41,A -85,B 0,C 180,E1 -3061.441,E2 -3061.441} C_VEL
LIN {X 0,Y 558.743,Z 753.998,A -85,B 0,C 180,E1 -3062.163,E2 -3062.163} C_VEL
LIN {X 0,Y 558.795,Z 753.18,A -85,B 0,C 180,E1 -3062.884,E2 -3062.884} C_VEL
LIN {X 0,Y 558.825,Z 751.961,A -85,B 0,C 180,E1 -3063.605,E2 -3063.605} C_VEL
LIN {X 0,Y 558.792,Z 749.357,A -85,B 0,C 180,E1 -3064.689,E2 -3064.689} C_VEL
LIN {X 0,Y 558.883,Z 745.704,A -85,B 0,C 180,E1 -3065.774,E2 -3065.774} C_VEL
LIN {X 0,Y 558.891,Z 740.987,A -85,B 0,C 180,E1 -3066.861,E2 -3066.861} C_VEL
LIN {X 0,Y 558.961,Z 734.953,A -85,B 0,C 180,E1 -3067.95,E2 -3067.95} C_VEL
LIN {X 0,Y 559.048,Z 727.481,A -85,B 0,C 180,E1 -3069.041,E2 -3069.041} C_VEL
LIN {X 0,Y 559.143,Z 719.837,A -85,B 0,C 180,E1 -3069.952,E2 -3069.952} C_VEL
LIN {X 0,Y 559.3,Z 710.516,A -85,B 0,C 180,E1 -3070.864,E2 -3070.864} C_VEL
LIN {X 0,Y 559.436,Z 700.204,A -85,B 0,C 180,E1 -3071.687,E2 -3071.687} C_VEL
LIN {X 0,Y 559.647,Z 688.738,A -85,B 0,C 180,E1 -3072.419,E2 -3072.419} C_VEL
LIN {X 0,Y 559.795,Z 676.606,A -85,B 0,C 180,E1 -3073.015,E2 -3073.015} C_VEL
LIN {X 0,Y 559.898,Z 663.907,A -85,B 0,C 180,E1 -3073.474,E2 -3073.474} C_VEL
LIN {X 0,Y 560.03,Z 650.748,A -85,B 0,C 180,E1 -3073.794,E2 -3073.794} C_VEL
LIN {X 0,Y 560.223,Z 547.056,A -85,B 0,C 180,E1 -3075.148,E2 -3075.148} C_VEL
LIN {X 0,Y 559.41,Z 541.829,A -85,B 0,C 180,E1 -3075.239,E2 -3075.239} C_VEL
LIN {X 0,Y 559.48,Z 536.223,A -85,B 0,C 180,E1 -3076,E2 -3076} C_VEL
LIN {X 0,Y 558.871,Z 532.774,A -85,B 0,C 180,E1 -3076.487,E2 -3076.487} C_VEL
LIN {X 0,Y 553.364,Z 522.131,A -85,B 0,C 180,E1 -3078.12,E2 -3078.12} C_VEL
LIN {X 0,Y 552.749,Z 518.706,A -85,B 0,C 180,E1 -3078.618,E2 -3078.618} C_VEL
LIN {X 0,Y 553.063,Z 500.04,A -85,B 0,C 180,E1 -3081.233,E2 -3081.233} C_VEL
LIN {X 0,Y 553.478,Z 480.743,A -85,B 0,C 180,E1 -3083.975,E2 -3083.975} C_VEL
LIN {X 0,Y 553.53,Z 473.919,A -85,B 0,C 180,E1 -3084.959,E2 -3084.959} C_VEL
LIN {X 0,Y 552.143,Z 466.833,A -85,B 0,C 180,E1 -3086.074,E2 -3086.074} C_VEL
LIN {X 0,Y 552.114,Z 466.834,A -85,B 0,C 180,E1 -3088.928,E2 -3088.928} C_VEL
LIN {X 0,Y 552.114,Z 466.839,A -85,B 0,C 180,E1 -3091.475,E2 -3091.475} C_VEL
LIN {X 0,Y 552.14,Z 466.83,A -85,B 0,C 180,E1 -3094.171,E2 -3094.171} C_VEL
LIN {X 0,Y 552.111,Z 466.831,A -85,B 0,C 180,E1 -3096.747,E2 -3096.747} C_VEL
LIN {X 0,Y 552.135,Z 466.837,A -85,B 0,C 180,E1 -3099.527,E2 -3099.527} C_VEL
LIN {X 0,Y 552.132,Z 466.828,A -85,B 0,C 180,E1 -3102.425,E2 -3102.425} C_VEL
LIN {X 0,Y 552.101,Z 466.842,A -85,B 0,C 180,E1 -3105.563,E2 -3105.563} C_VEL
LIN {X 0,Y 552.133,Z 466.828,A -85,B 0,C 180,E1 -3108.555,E2 -3108.555} C_VEL
LIN {X 0,Y 552.12,Z 466.837,A -85,B 0,C 180,E1 -3111.411,E2 -3111.411} C_VEL
LIN {X 0,Y 552.088,Z 466.835,A -85,B 0,C 180,E1 -3114.156,E2 -3114.156} C_VEL
LIN {X 0,Y 552.118,Z 466.831,A -85,B 0,C 180,E1 -3116.814,E2 -3116.814} C_VEL
LIN {X 0,Y 552.105,Z 466.839,A -85,B 0,C 180,E1 -3119.391,E2 -3119.391} C_VEL
LIN {X 0,Y 552.112,Z 466.835,A -85,B 0,C 180,E1 -3121.902,E2 -3121.902} C_VEL
LIN {X 0,Y 552.158,Z 466.825,A -85,B 0,C 180,E1 -3124.649,E2 -3124.649} C_VEL
LIN {X 0,Y 552.094,Z 466.843,A -85,B 0,C 180,E1 -3127.549,E2 -3127.549} C_VEL
LIN {X 0,Y 552.152,Z 466.826,A -85,B 0,C 180,E1 -3130.373,E2 -3130.373} C_VEL
LIN {X 0,Y 552.158,Z 466.827,A -85,B 0,C 180,E1 -3132.977,E2 -3132.977} C_VEL
LIN {X 0,Y 552.139,Z 466.83,A -85,B 0,C 180,E1 -3136.004,E2 -3136.004} C_VEL
LIN {X 0,Y 552.166,Z 466.827,A -85,B 0,C 180,E1 -3138.993,E2 -3138.993} C_VEL
LIN {X 0,Y 552.166,Z 466.827,A -85,B 0,C 180,E1 -3141.952,E2 -3141.952} C_VEL
LIN {X 0,Y 552.232,Z 466.818,A -85,B 0,C 180,E1 -3144.889,E2 -3144.889} C_VEL
LIN {X 0,Y 552.229,Z 466.82,A -85,B 0,C 180,E1 -3147.812,E2 -3147.812} C_VEL
LIN {X 0,Y 552.243,Z 466.815,A -85,B 0,C 180,E1 -3150.729,E2 -3150.729} C_VEL
LIN {X 0,Y 552.208,Z 466.821,A -85,B 0,C 180,E1 -3152.918,E2 -3152.918} C_VEL
LIN {X 0,Y 552.205,Z 466.823,A -85,B 0,C 180,E1 -3155.844,E2 -3155.844} C_VEL
LIN {X 0,Y 552.16,Z 466.826,A -85,B 0,C 180,E1 -3158.786,E2 -3158.786} C_VEL
LIN {X 0,Y 552.165,Z 466.829,A -85,B 0,C 180,E1 -3161.75,E2 -3161.75} C_VEL
LIN {X 0,Y 552.139,Z 466.829,A -85,B 0,C 180,E1 -3164.748,E2 -3164.748} C_VEL
LIN {X 0,Y 552.112,Z 466.834,A -85,B 0,C 180,E1 -3167.788,E2 -3167.788} C_VEL
LIN {X 0,Y 552.133,Z 466.829,A -85,B 0,C 180,E1 -3170.101,E2 -3170.101} C_VEL
LIN {X 0,Y 552.098,Z 466.832,A -85,B 0,C 180,E1 -3172.451,E2 -3172.451} C_VEL
LIN {X 0,Y 552.158,Z 466.835,A -85,B 0,C 180,E1 -3175.35,E2 -3175.35} C_VEL
LIN {X 0,Y 552.122,Z 466.83,A -85,B 0,C 180,E1 -3178.098,E2 -3178.098} C_VEL
LIN {X 0,Y 552.107,Z 466.832,A -85,B 0,C 180,E1 -3180.609,E2 -3180.609} C_VEL
LIN {X 0,Y 552.118,Z 466.837,A -85,B 0,C 180,E1 -3183.186,E2 -3183.186} C_VEL
LIN {X 0,Y 552.087,Z 466.836,A -85,B 0,C 180,E1 -3185.844,E2 -3185.844} C_VEL
LIN {X 0,Y 552.127,Z 466.834,A -85,B 0,C 180,E1 -3189.062,E2 -3189.062} C_VEL
LIN {X 0,Y 552.143,Z 466.835,A -85,B 0,C 180,E1 -3191.444,E2 -3191.444} C_VEL
LIN {X 0,Y 552.097,Z 466.833,A -85,B 0,C 180,E1 -3194.532,E2 -3194.532} C_VEL
LIN {X 0,Y 552.132,Z 466.834,A -85,B 0,C 180,E1 -3197.585,E2 -3197.585} C_VEL
LIN {X 0,Y 552.136,Z 466.828,A -85,B 0,C 180,E1 -3200.473,E2 -3200.473} C_VEL
LIN {X 0,Y 552.109,Z 466.841,A -85,B 0,C 180,E1 -3203.317,E2 -3203.317} C_VEL
LIN {X 0,Y 552.132,Z 466.829,A -85,B 0,C 180,E1 -3205.939,E2 -3205.939} C_VEL
LIN {X 0,Y 552.122,Z 466.831,A -85,B 0,C 180,E1 -3208.541,E2 -3208.541} C_VEL
LIN {X 0,Y 552.128,Z 466.837,A -85,B 0,C 180,E1 -3211.438,E2 -3211.438} C_VEL
LIN {X 0,Y 552.134,Z 466.832,A -85,B 0,C 180,E1 -3214.356,E2 -3214.356} C_VEL
LIN {X 0,Y 552.177,Z 466.969,A -85,B 0,C 180,E1 -3214.934,E2 -3214.934} C_VEL
LIN {X 0,Y 553.598,Z 474.928,A -85,B 0,C 180,E1 -3216.072,E2 -3216.072} C_VEL
LIN {X 0,Y 553.261,Z 494.395,A -85,B 0,C 180,E1 -3218.775,E2 -3218.775} C_VEL
LIN {X 0,Y 552.92,Z 513.96,A -85,B 0,C 180,E1 -3221.472,E2 -3221.472} C_VEL
LIN {X 0,Y 552.54,Z 536.17,A -85,B 0,C 180,E1 -3224.508,E2 -3224.508} C_VEL
LIN {X 0,Y 552.47,Z 544.899,A -85,B 0,C 180,E1 -3225.672,E2 -3225.672} C_VEL
LIN {X 0,Y 553.417,Z 551.154,A -85,B 0,C 180,E1 -3225.78,E2 -3225.78} C_VEL
LIN {X 0,Y 553.153,Z 653.217,A -85,B 0,C 180,E1 -3227.13,E2 -3227.13} C_VEL
LIN {X 0,Y 553.035,Z 664.33,A -85,B 0,C 180,E1 -3227.384,E2 -3227.384} C_VEL
LIN {X 0,Y 552.858,Z 677.814,A -85,B 0,C 180,E1 -3227.846,E2 -3227.846} C_VEL
LIN {X 0,Y 552.682,Z 689.371,A -85,B 0,C 180,E1 -3228.4,E2 -3228.4} C_VEL
LIN {X 0,Y 552.536,Z 699.313,A -85,B 0,C 180,E1 -3229.001,E2 -3229.001} C_VEL
LIN {X 0,Y 552.366,Z 709.3,A -85,B 0,C 180,E1 -3229.739,E2 -3229.739} C_VEL
LIN {X 0,Y 552.175,Z 719.415,A -85,B 0,C 180,E1 -3230.661,E2 -3230.661} C_VEL
LIN {X 0,Y 552.042,Z 727.615,A -85,B 0,C 180,E1 -3231.581,E2 -3231.581} C_VEL
LIN {X 0,Y 551.913,Z 735.609,A -85,B 0,C 180,E1 -3232.684,E2 -3232.684} C_VEL
LIN {X 0,Y 551.811,Z 741.344,A -85,B 0,C 180,E1 -3233.65,E2 -3233.65} C_VEL
LIN {X 0,Y 551.803,Z 745.632,A -85,B 0,C 180,E1 -3234.519,E2 -3234.519} C_VEL
LIN {X 0,Y 551.766,Z 749.979,A -85,B 0,C 180,E1 -3235.617,E2 -3235.617} C_VEL
LIN {X 0,Y 551.751,Z 752.343,A -85,B 0,C 180,E1 -3236.348,E2 -3236.348} C_VEL
LIN {X 0,Y 551.724,Z 754.18,A -85,B 0,C 180,E1 -3237.079,E2 -3237.079} C_VEL
LIN {X 0,Y 551.645,Z 756.643,A -85,B 0,C 180,E1 -3238.54,E2 -3238.54} C_VEL
LIN {X 0,Y 551.642,Z 757.254,A -85,B 0,C 180,E1 -3239.27,E2 -3239.27} C_VEL
LIN {X 0,Y 551.642,Z 757.31,A -85,B 0,C 180,E1 -3240.73,E2 -3240.73} C_VEL
LIN {X 0,Y 551.645,Z 756.735,A -85,B 0,C 180,E1 -3241.46,E2 -3241.46} C_VEL
LIN {X 0,Y 551.724,Z 754.396,A -85,B 0,C 180,E1 -3242.921,E2 -3242.921} C_VEL
LIN {X 0,Y 551.764,Z 751.521,A -85,B 0,C 180,E1 -3244.017,E2 -3244.017} C_VEL
LIN {X 0,Y 551.723,Z 747.609,A -85,B 0,C 180,E1 -3245.116,E2 -3245.116} C_VEL
LIN {X 0,Y 551.836,Z 743.171,A -85,B 0,C 180,E1 -3246.098,E2 -3246.098} C_VEL
LIN {X 0,Y 551.885,Z 737.375,A -85,B 0,C 180,E1 -3247.132,E2 -3247.132} C_VEL
LIN {X 0,Y 551.983,Z 731.143,A -85,B 0,C 180,E1 -3248.051,E2 -3248.051} C_VEL
LIN {X 0,Y 552.102,Z 723.638,A -85,B 0,C 180,E1 -3248.971,E2 -3248.971} C_VEL
LIN {X 0,Y 552.229,Z 716.535,A -85,B 0,C 180,E1 -3249.708,E2 -3249.708} C_VEL
LIN {X 0,Y 552.393,Z 708.093,A -85,B 0,C 180,E1 -3250.446,E2 -3250.446} C_VEL
LIN {X 0,Y 552.547,Z 698.403,A -85,B 0,C 180,E1 -3251.15,E2 -3251.15} C_VEL
LIN {X 0,Y 552.737,Z 686.774,A -85,B 0,C 180,E1 -3251.831,E2 -3251.831} C_VEL
LIN {X 0,Y 552.899,Z 674.123,A -85,B 0,C 180,E1 -3252.386,E2 -3252.386} C_VEL
LIN {X 0,Y 553.028,Z 662.427,A -85,B 0,C 180,E1 -3252.756,E2 -3252.756} C_VEL
LIN {X 0,Y 553.125,Z 651.679,A -85,B 0,C 180,E1 -3252.987,E2 -3252.987} C_VEL
LIN {X 0,Y 553.362,Z 550.858,A -85,B 0,C 180,E1 -3254.316,E2 -3254.316} C_VEL
LIN {X 0,Y 552.444,Z 544.73,A -85,B 0,C 180,E1 -3254.422,E2 -3254.422} C_VEL
LIN {X 0,Y 552.752,Z 522.905,A -85,B 0,C 180,E1 -3257.39,E2 -3257.39} C_VEL
LIN {X 0,Y 553.099,Z 502.096,A -85,B 0,C 180,E1 -3260.258,E2 -3260.258} C_VEL
LIN {X 0,Y 553.441,Z 478.764,A -85,B 0,C 180,E1 -3263.373,E2 -3263.373} C_VEL
LIN {X 0,Y 553.319,Z 472.799,A -85,B 0,C 180,E1 -3264.181,E2 -3264.181} C_VEL
LIN {X 0,Y 552.167,Z 466.833,A -85,B 0,C 180,E1 -3265.066,E2 -3265.066} C_VEL
LIN {X 0,Y 552.112,Z 466.835,A -85,B 0,C 180,E1 -3268.098,E2 -3268.098} C_VEL
LIN {X 0,Y 552.105,Z 466.841,A -85,B 0,C 180,E1 -3270.609,E2 -3270.609} C_VEL
LIN {X 0,Y 552.118,Z 466.835,A -85,B 0,C 180,E1 -3273.186,E2 -3273.186} C_VEL
LIN {X 0,Y 552.089,Z 466.836,A -85,B 0,C 180,E1 -3275.843,E2 -3275.843} C_VEL
LIN {X 0,Y 552.128,Z 466.833,A -85,B 0,C 180,E1 -3279.062,E2 -3279.062} C_VEL
LIN {X 0,Y 552.123,Z 466.831,A -85,B 0,C 180,E1 -3281.446,E2 -3281.446} C_VEL
LIN {X 0,Y 552.096,Z 466.843,A -85,B 0,C 180,E1 -3284.532,E2 -3284.532} C_VEL
LIN {X 0,Y 552.134,Z 466.829,A -85,B 0,C 180,E1 -3287.584,E2 -3287.584} C_VEL
LIN {X 0,Y 552.132,Z 466.837,A -85,B 0,C 180,E1 -3290.473,E2 -3290.473} C_VEL
LIN {X 0,Y 552.117,Z 466.831,A -85,B 0,C 180,E1 -3293.316,E2 -3293.316} C_VEL
LIN {X 0,Y 552.131,Z 466.833,A -85,B 0,C 180,E1 -3295.939,E2 -3295.939} C_VEL
LIN {X 0,Y 552.121,Z 466.838,A -85,B 0,C 180,E1 -3298.541,E2 -3298.541} C_VEL
LIN {X 0,Y 552.127,Z 466.831,A -85,B 0,C 180,E1 -3301.438,E2 -3301.438} C_VEL
LIN {X 0,Y 552.133,Z 466.839,A -85,B 0,C 180,E1 -3304.356,E2 -3304.356} C_VEL
LIN {X 0,Y 552.145,Z 466.976,A -85,B 0,C 180,E1 -3305.614,E2 -3305.614} C_VEL
LIN {X 0,Y 553.897,Z 474.909,A -85,B 0,C 180,E1 -3306.685,E2 -3306.685} C_VEL
LIN {X 0,Y 553.413,Z 496.903,A -85,B 0,C 180,E1 -3309.365,E2 -3309.365} C_VEL
LIN {X 0,Y 552.965,Z 522.29,A -85,B 0,C 180,E1 -3312.407,E2 -3312.407} C_VEL
LIN {X 0,Y 552.952,Z 523.795,A -85,B 0,C 180,E1 -3312.581,E2 -3312.581} C_VEL
LIN {X 0,Y 554.253,Z 532.388,A -85,B 0,C 180,E1 -3312.737,E2 -3312.737} C_VEL
LIN {X 0,Y 553.759,Z 662.882,A -85,B 0,C 180,E1 -3314.472,E2 -3314.472} C_VEL
LIN {X 0,Y 553.566,Z 677.208,A -85,B 0,C 180,E1 -3314.815,E2 -3314.815} C_VEL
LIN {X 0,Y 553.379,Z 690.706,A -85,B 0,C 180,E1 -3315.285,E2 -3315.285} C_VEL
LIN {X 0,Y 553.155,Z 704.64,A -85,B 0,C 180,E1 -3315.937,E2 -3315.937} C_VEL
LIN {X 0,Y 552.865,Z 717.102,A -85,B 0,C 180,E1 -3316.679,E2 -3316.679} C_VEL
LIN {X 0,Y 552.618,Z 729.645,A -85,B 0,C 180,E1 -3317.607,E2 -3317.607} C_VEL
LIN {X 0,Y 552.451,Z 740.274,A -85,B 0,C 180,E1 -3318.571,E2 -3318.571} C_VEL
LIN {X 0,Y 552.179,Z 750.852,A -85,B 0,C 180,E1 -3319.736,E2 -3319.736} C_VEL
LIN {X 0,Y 552.033,Z 759.174,A -85,B 0,C 180,E1 -3320.843,E2 -3320.843} C_VEL
LIN {X 0,Y 551.913,Z 767.128,A -85,B 0,C 180,E1 -3322.132,E2 -3322.132} C_VEL
LIN {X 0,Y 551.822,Z 773.528,A -85,B 0,C 180,E1 -3323.418,E2 -3323.418} C_VEL
LIN {X 0,Y 551.792,Z 777.961,A -85,B 0,C 180,E1 -3324.518,E2 -3324.518} C_VEL
LIN {X 0,Y 551.759,Z 781.444,A -85,B 0,C 180,E1 -3325.617,E2 -3325.617} C_VEL
LIN {X 0,Y 551.72,Z 784.832,A -85,B 0,C 180,E1 -3327.079,E2 -3327.079} C_VEL
LIN {X 0,Y 551.64,Z 786.833,A -85,B 0,C 180,E1 -3328.54,E2 -3328.54} C_VEL
LIN {X 0,Y 551.639,Z 787.5,A -85,B 0,C 180,E1 -3330,E2 -3330} C_VEL
LIN {X 0,Y 551.64,Z 786.834,A -85,B 0,C 180,E1 -3331.46,E2 -3331.46} C_VEL
LIN {X 0,Y 551.72,Z 784.834,A -85,B 0,C 180,E1 -3332.921,E2 -3332.921} C_VEL
LIN {X 0,Y 551.759,Z 781.446,A -85,B 0,C 180,E1 -3334.383,E2 -3334.383} C_VEL
LIN {X 0,Y 551.825,Z 776.568,A -85,B 0,C 180,E1 -3335.848,E2 -3335.848} C_VEL
LIN {X 0,Y 551.833,Z 770.053,A -85,B 0,C 180,E1 -3337.317,E2 -3337.317} C_VEL
LIN {X 0,Y 551.963,Z 762.801,A -85,B 0,C 180,E1 -3338.604,E2 -3338.604} C_VEL
LIN {X 0,Y 552.116,Z 753.821,A -85,B 0,C 180,E1 -3339.895,E2 -3339.895} C_VEL
LIN {X 0,Y 552.346,Z 744.391,A -85,B 0,C 180,E1 -3341.003,E2 -3341.003} C_VEL
LIN {X 0,Y 552.539,Z 733.952,A -85,B 0,C 180,E1 -3342.022,E2 -3342.022} C_VEL
LIN {X 0,Y 552.76,Z 722.431,A -85,B 0,C 180,E1 -3342.95,E2 -3342.95} C_VEL
LIN {X 0,Y 553.032,Z 709.639,A -85,B 0,C 180,E1 -3343.785,E2 -3343.785} C_VEL
LIN {X 0,Y 553.301,Z 697.146,A -85,B 0,C 180,E1 -3344.435,E2 -3344.435} C_VEL
LIN {X 0,Y 553.485,Z 683.984,A -85,B 0,C 180,E1 -3344.967,E2 -3344.967} C_VEL
LIN {X 0,Y 553.655,Z 669.881,A -85,B 0,C 180,E1 -3345.381,E2 -3345.381} C_VEL
LIN {X 0,Y 553.782,Z 655.591,A -85,B 0,C 180,E1 -3345.645,E2 -3345.645} C_VEL
LIN {X 0,Y 554.178,Z 530.944,A -85,B 0,C 180,E1 -3347.284,E2 -3347.284} C_VEL
LIN {X 0,Y 552.954,Z 523.587,A -85,B 0,C 180,E1 -3347.439,E2 -3347.439} C_VEL
LIN {X 0,Y 553.354,Z 500.101,A -85,B 0,C 180,E1 -3350.249,E2 -3350.249} C_VEL
LIN {X 0,Y 553.908,Z 476.182,A -85,B 0,C 180,E1 -3353.162,E2 -3353.162} C_VEL
LIN {X 0,Y 553.428,Z 472.429,A -85,B 0,C 180,E1 -3353.651,E2 -3353.651} C_VEL
LIN {X 0,Y 552.147,Z 466.833,A -85,B 0,C 180,E1 -3354.436,E2 -3354.436} C_VEL
LIN {X 0,Y 552.142,Z 466.835,A -85,B 0,C 180,E1 -3357.273,E2 -3357.273} C_VEL
LIN {X 0,Y 552.122,Z 466.836,A -85,B 0,C 180,E1 -3360.051,E2 -3360.051} C_VEL
LIN {X 0,Y 552.119,Z 466.834,A -85,B 0,C 180,E1 -3362.847,E2 -3362.847} C_VEL
LIN {X 0,Y 552.079,Z 466.845,A -85,B 0,C 180,E1 -3365.44,E2 -3365.44} C_VEL
LIN {X 0,Y 552.099,Z 466.837,A -85,B 0,C 180,E1 -3367.886,E2 -3367.886} C_VEL
LIN {X 0,Y 552.112,Z 466.833,A -85,B 0,C 180,E1 -3370.481,E2 -3370.481} C_VEL
LIN {X 0,Y 552.118,Z 466.836,A -85,B 0,C 180,E1 -3373.484,E2 -3373.484} C_VEL
LIN {X 0,Y 552.109,Z 466.835,A -85,B 0,C 180,E1 -3376.576,E2 -3376.576} C_VEL
LIN {X 0,Y 552.123,Z 466.834,A -85,B 0,C 180,E1 -3379.52,E2 -3379.52} C_VEL
LIN {X 0,Y 552.097,Z 466.837,A -85,B 0,C 180,E1 -3382.336,E2 -3382.336} C_VEL
LIN {X 0,Y 552.12,Z 466.838,A -85,B 0,C 180,E1 -3385.054,E2 -3385.054} C_VEL
LIN {X 0,Y 552.131,Z 466.831,A -85,B 0,C 180,E1 -3387.682,E2 -3387.682} C_VEL
LIN {X 0,Y 552.117,Z 466.837,A -85,B 0,C 180,E1 -3390.235,E2 -3390.235} C_VEL
LIN {X 0,Y 552.144,Z 466.837,A -85,B 0,C 180,E1 -3393,E2 -3393} C_VEL
LIN {X 0,Y 552.118,Z 466.837,A -85,B 0,C 180,E1 -3395.161,E2 -3395.161} C_VEL
LIN {X 0,Y 552.147,Z 466.851,A -85,B 0,C 180,E1 -3396.055,E2 -3396.055} C_VEL
LIN {X 0,Y 553.562,Z 474.395,A -85,B 0,C 180,E1 -3397.218,E2 -3397.218} C_VEL
LIN {X 0,Y 553.176,Z 493.493,A -85,B 0,C 180,E1 -3399.938,E2 -3399.938} C_VEL
LIN {X 0,Y 552.859,Z 514.294,A -85,B 0,C 180,E1 -3402.858,E2 -3402.858} C_VEL
LIN {X 0,Y 552.483,Z 537.07,A -85,B 0,C 180,E1 -3406.013,E2 -3406.013} C_VEL
LIN {X 0,Y 552.424,Z 541.835,A -85,B 0,C 180,E1 -3406.668,E2 -3406.668} C_VEL
LIN {X 0,Y 553.413,Z 548.644,A -85,B 0,C 180,E1 -3406.786,E2 -3406.786} C_VEL
LIN {X 0,Y 553.116,Z 651.369,A -85,B 0,C 180,E1 -3408.145,E2 -3408.145} C_VEL
LIN {X 0,Y 552.97,Z 664.5,A -85,B 0,C 180,E1 -3408.476,E2 -3408.476} C_VEL
LIN {X 0,Y 552.827,Z 677.43,A -85,B 0,C 180,E1 -3408.96,E2 -3408.96} C_VEL
LIN {X 0,Y 552.706,Z 689.305,A -85,B 0,C 180,E1 -3409.56,E2 -3409.56} C_VEL
LIN {X 0,Y 552.418,Z 700.629,A -85,B 0,C 180,E1 -3410.295,E2 -3410.295} C_VEL
LIN {X 0,Y 552.322,Z 710.779,A -85,B 0,C 180,E1 -3411.125,E2 -3411.125} C_VEL
LIN {X 0,Y 552.078,Z 720.806,A -85,B 0,C 180,E1 -3412.134,E2 -3412.134} C_VEL
LIN {X 0,Y 551.983,Z 728.558,A -85,B 0,C 180,E1 -3413.089,E2 -3413.089} C_VEL
LIN {X 0,Y 551.918,Z 735.565,A -85,B 0,C 180,E1 -3414.153,E2 -3414.153} C_VEL
LIN {X 0,Y 551.809,Z 741.435,A -85,B 0,C 180,E1 -3415.251,E2 -3415.251} C_VEL
LIN {X 0,Y 551.776,Z 746.069,A -85,B 0,C 180,E1 -3416.349,E2 -3416.349} C_VEL
LIN {X 0,Y 551.721,Z 749.599,A -85,B 0,C 180,E1 -3417.445,E2 -3417.445} C_VEL
LIN {X 0,Y 551.649,Z 752.139,A -85,B 0,C 180,E1 -3418.54,E2 -3418.54} C_VEL
LIN {X 0,Y 551.642,Z 753.305,A -85,B 0,C 180,E1 -3419.27,E2 -3419.27} C_VEL
LIN {X 0,Y 551.642,Z 754.07,A -85,B 0,C 180,E1 -3420,E2 -3420} C_VEL
LIN {X 0,Y 551.644,Z 754.403,A -85,B 0,C 180,E1 -3421.46,E2 -3421.46} C_VEL
LIN {X 0,Y 551.654,Z 753.983,A -85,B 0,C 180,E1 -3422.19,E2 -3422.19} C_VEL
LIN {X 0,Y 551.72,Z 753.158,A -85,B 0,C 180,E1 -3422.921,E2 -3422.921} C_VEL
LIN {X 0,Y 551.738,Z 751.931,A -85,B 0,C 180,E1 -3423.652,E2 -3423.652} C_VEL
LIN {X 0,Y 551.693,Z 749.32,A -85,B 0,C 180,E1 -3424.75,E2 -3424.75} C_VEL
LIN {X 0,Y 551.796,Z 745.65,A -85,B 0,C 180,E1 -3425.848,E2 -3425.848} C_VEL
LIN {X 0,Y 551.819,Z 740.921,A -85,B 0,C 180,E1 -3426.949,E2 -3426.949} C_VEL
LIN {X 0,Y 551.891,Z 734.868,A -85,B 0,C 180,E1 -3428.052,E2 -3428.052} C_VEL
LIN {X 0,Y 552.002,Z 727.371,A -85,B 0,C 180,E1 -3429.157,E2 -3429.157} C_VEL
LIN {X 0,Y 552.104,Z 719.716,A -85,B 0,C 180,E1 -3430.08,E2 -3430.08} C_VEL
LIN {X 0,Y 552.291,Z 710.359,A -85,B 0,C 180,E1 -3431.004,E2 -3431.004} C_VEL
LIN {X 0,Y 552.454,Z 700.003,A -85,B 0,C 180,E1 -3431.837,E2 -3431.837} C_VEL
LIN {X 0,Y 552.663,Z 688.499,A -85,B 0,C 180,E1 -3432.578,E2 -3432.578} C_VEL
LIN {X 0,Y 552.822,Z 676.289,A -85,B 0,C 180,E1 -3433.182,E2 -3433.182} C_VEL
LIN {X 0,Y 552.972,Z 663.443,A -85,B 0,C 180,E1 -3433.646,E2 -3433.646} C_VEL
LIN {X 0,Y 553.113,Z 651.29,A -85,B 0,C 180,E1 -3433.947,E2 -3433.947} C_VEL
LIN {X 0,Y 553.337,Z 547.953,A -85,B 0,C 180,E1 -3435.315,E2 -3435.315} C_VEL
LIN {X 0,Y 552.39,Z 541.812,A -85,B 0,C 180,E1 -3435.426,E2 -3435.426} C_VEL
LIN {X 0,Y 552.756,Z 520.682,A -85,B 0,C 180,E1 -3438.342,E2 -3438.342} C_VEL
LIN {X 0,Y 552.749,Z 518.706,A -85,B 0,C 180,E1 -3438.618,E2 -3438.618} C_VEL
LIN {X 0,Y 552.134,Z 515.302,A -85,B 0,C 180,E1 -3439.115,E2 -3439.115} C_VEL
LIN {X 0,Y 546.7,Z 504.864,A -85,B 0,C 180,E1 -3440.785,E2 -3440.785} C_VEL
LIN {X 0,Y 546.142,Z 501.474,A -85,B 0,C 180,E1 -3441.292,E2 -3441.292} C_VEL
LIN {X 0,Y 546.59,Z 482.041,A -85,B 0,C 180,E1 -3444.088,E2 -3444.088} C_VEL
LIN {X 0,Y 546.594,Z 475.07,A -85,B 0,C 180,E1 -3445.107,E2 -3445.107} C_VEL
LIN {X 0,Y 545.094,Z 467.712,A -85,B 0,C 180,E1 -3446.283,E2 -3446.283} C_VEL
LIN {X 0,Y 545.068,Z 467.717,A -85,B 0,C 180,E1 -3449.338,E2 -3449.338} C_VEL
LIN {X 0,Y 545.058,Z 467.716,A -85,B 0,C 180,E1 -3451.915,E2 -3451.915} C_VEL
LIN {X 0,Y 545.081,Z 467.708,A -85,B 0,C 180,E1 -3454.563,E2 -3454.563} C_VEL
LIN {X 0,Y 545.04,Z 467.717,A -85,B 0,C 180,E1 -3457.304,E2 -3457.304} C_VEL
LIN {X 0,Y 545.071,Z 467.71,A -85,B 0,C 180,E1 -3460.142,E2 -3460.142} C_VEL
LIN {X 0,Y 545.081,Z 467.709,A -85,B 0,C 180,E1 -3463.106,E2 -3463.106} C_VEL
LIN {X 0,Y 545.07,Z 467.709,A -85,B 0,C 180,E1 -3466.224,E2 -3466.224} C_VEL
LIN {X 0,Y 545.089,Z 467.707,A -85,B 0,C 180,E1 -3468.886,E2 -3468.886} C_VEL
LIN {X 0,Y 545.055,Z 467.716,A -85,B 0,C 180,E1 -3471.763,E2 -3471.763} C_VEL
LIN {X 0,Y 545.038,Z 467.712,A -85,B 0,C 180,E1 -3474.531,E2 -3474.531} C_VEL
LIN {X 0,Y 545.072,Z 467.712,A -85,B 0,C 180,E1 -3477.211,E2 -3477.211} C_VEL
LIN {X 0,Y 545.066,Z 467.714,A -85,B 0,C 180,E1 -3479.81,E2 -3479.81} C_VEL
LIN {X 0,Y 545.083,Z 467.707,A -85,B 0,C 180,E1 -3482.344,E2 -3482.344} C_VEL
LIN {X 0,Y 545.12,Z 467.703,A -85,B 0,C 180,E1 -3484.82,E2 -3484.82} C_VEL
LIN {X 0,Y 545.039,Z 467.717,A -85,B 0,C 180,E1 -3487.242,E2 -3487.242} C_VEL
LIN {X 0,Y 545.123,Z 467.701,A -85,B 0,C 180,E1 -3490.415,E2 -3490.415} C_VEL
LIN {X 0,Y 545.078,Z 467.717,A -85,B 0,C 180,E1 -3493.521,E2 -3493.521} C_VEL
LIN {X 0,Y 545.098,Z 467.709,A -85,B 0,C 180,E1 -3495.82,E2 -3495.82} C_VEL
LIN {X 0,Y 545.121,Z 467.703,A -85,B 0,C 180,E1 -3498.849,E2 -3498.849} C_VEL
LIN {X 0,Y 545.136,Z 467.704,A -85,B 0,C 180,E1 -3501.847,E2 -3501.847} C_VEL
LIN {X 0,Y 545.207,Z 467.692,A -85,B 0,C 180,E1 -3504.823,E2 -3504.823} C_VEL
LIN {X 0,Y 545.2,Z 467.696,A -85,B 0,C 180,E1 -3507.784,E2 -3507.784} C_VEL
LIN {X 0,Y 545.214,Z 467.691,A -85,B 0,C 180,E1 -3510.739,E2 -3510.739} C_VEL
LIN {X 0,Y 545.175,Z 467.698,A -85,B 0,C 180,E1 -3512.956,E2 -3512.956} C_VEL
LIN {X 0,Y 545.175,Z 467.698,A -85,B 0,C 180,E1 -3515.919,E2 -3515.919} C_VEL
LIN {X 0,Y 545.12,Z 467.704,A -85,B 0,C 180,E1 -3518.9,E2 -3518.9} C_VEL
LIN {X 0,Y 545.138,Z 467.702,A -85,B 0,C 180,E1 -3521.904,E2 -3521.904} C_VEL
LIN {X 0,Y 545.088,Z 467.709,A -85,B 0,C 180,E1 -3524.944,E2 -3524.944} C_VEL
LIN {X 0,Y 545.08,Z 467.708,A -85,B 0,C 180,E1 -3528.026,E2 -3528.026} C_VEL
LIN {X 0,Y 545.097,Z 467.704,A -85,B 0,C 180,E1 -3530.372,E2 -3530.372} C_VEL
LIN {X 0,Y 545.094,Z 467.712,A -85,B 0,C 180,E1 -3533.559,E2 -3533.559} C_VEL
LIN {X 0,Y 545.082,Z 467.708,A -85,B 0,C 180,E1 -3536.001,E2 -3536.001} C_VEL
LIN {X 0,Y 545.091,Z 467.707,A -85,B 0,C 180,E1 -3538.748,E2 -3538.748} C_VEL
LIN {X 0,Y 545.06,Z 467.714,A -85,B 0,C 180,E1 -3541.679,E2 -3541.679} C_VEL
LIN {X 0,Y 545.064,Z 467.709,A -85,B 0,C 180,E1 -3544.564,E2 -3544.564} C_VEL
LIN {X 0,Y 545.04,Z 467.721,A -85,B 0,C 180,E1 -3547.304,E2 -3547.304} C_VEL
LIN {X 0,Y 545.074,Z 467.708,A -85,B 0,C 180,E1 -3550.142,E2 -3550.142} C_VEL
LIN {X 0,Y 545.089,Z 467.712,A -85,B 0,C 180,E1 -3553.106,E2 -3553.106} C_VEL
LIN {X 0,Y 545.051,Z 467.71,A -85,B 0,C 180,E1 -3556.226,E2 -3556.226} C_VEL
LIN {X 0,Y 545.083,Z 467.71,A -85,B 0,C 180,E1 -3558.886,E2 -3558.886} C_VEL
LIN {X 0,Y 545.086,Z 467.709,A -85,B 0,C 180,E1 -3560.819,E2 -3560.819} C_VEL
LIN {X 0,Y 545.045,Z 467.716,A -85,B 0,C 180,E1 -3563.62,E2 -3563.62} C_VEL
LIN {X 0,Y 545.07,Z 467.708,A -85,B 0,C 180,E1 -3566.328,E2 -3566.328} C_VEL
LIN {X 0,Y 545.069,Z 467.714,A -85,B 0,C 180,E1 -3568.952,E2 -3568.952} C_VEL
LIN {X 0,Y 545.104,Z 467.711,A -85,B 0,C 180,E1 -3571.508,E2 -3571.508} C_VEL
LIN {X 0,Y 545.132,Z 467.707,A -85,B 0,C 180,E1 -3574.657,E2 -3574.657} C_VEL
LIN {X 0,Y 545.154,Z 467.91,A -85,B 0,C 180,E1 -3574.781,E2 -3574.781} C_VEL
LIN {X 0,Y 546.618,Z 475.634,A -85,B 0,C 180,E1 -3575.905,E2 -3575.905} C_VEL
LIN {X 0,Y 546.402,Z 489.538,A -85,B 0,C 180,E1 -3577.833,E2 -3577.833} C_VEL
LIN {X 0,Y 546.028,Z 511.058,A -85,B 0,C 180,E1 -3580.84,E2 -3580.84} C_VEL
LIN {X 0,Y 545.645,Z 532.01,A -85,B 0,C 180,E1 -3583.731,E2 -3583.731} C_VEL
LIN {X 0,Y 545.468,Z 544.744,A -85,B 0,C 180,E1 -3585.482,E2 -3585.482} C_VEL
LIN {X 0,Y 546.537,Z 552.903,A -85,B 0,C 180,E1 -3585.619,E2 -3585.619} C_VEL
LIN {X 0,Y 546.243,Z 653.208,A -85,B 0,C 180,E1 -3586.964,E2 -3586.964} C_VEL
LIN {X 0,Y 546.102,Z 664.328,A -85,B 0,C 180,E1 -3587.221,E2 -3587.221} C_VEL
LIN {X 0,Y 545.937,Z 677.818,A -85,B 0,C 180,E1 -3587.689,E2 -3587.689} C_VEL
LIN {X 0,Y 545.722,Z 688.83,A -85,B 0,C 180,E1 -3588.22,E2 -3588.22} C_VEL
LIN {X 0,Y 545.585,Z 698.278,A -85,B 0,C 180,E1 -3588.789,E2 -3588.789} C_VEL
LIN {X 0,Y 545.423,Z 706.957,A -85,B 0,C 180,E1 -3589.419,E2 -3589.419} C_VEL
LIN {X 0,Y 545.222,Z 715.568,A -85,B 0,C 180,E1 -3590.166,E2 -3590.166} C_VEL
LIN {X 0,Y 545.063,Z 724.498,A -85,B 0,C 180,E1 -3591.099,E2 -3591.099} C_VEL
LIN {X 0,Y 544.897,Z 733.198,A -85,B 0,C 180,E1 -3592.217,E2 -3592.217} C_VEL
LIN {X 0,Y 544.761,Z 740.496,A -85,B 0,C 180,E1 -3593.407,E2 -3593.407} C_VEL
LIN {X 0,Y 544.74,Z 745.627,A -85,B 0,C 180,E1 -3594.447,E2 -3594.447} C_VEL
LIN {X 0,Y 544.664,Z 749.975,A -85,B 0,C 180,E1 -3595.56,E2 -3595.56} C_VEL
LIN {X 0,Y 544.669,Z 752.344,A -85,B 0,C 180,E1 -3596.301,E2 -3596.301} C_VEL
LIN {X 0,Y 544.65,Z 754.179,A -85,B 0,C 180,E1 -3597.041,E2 -3597.041} C_VEL
LIN {X 0,Y 544.546,Z 756.645,A -85,B 0,C 180,E1 -3598.521,E2 -3598.521} C_VEL
LIN {X 0,Y 544.542,Z 757.252,A -85,B 0,C 180,E1 -3599.261,E2 -3599.261} C_VEL
LIN {X 0,Y 544.542,Z 757.309,A -85,B 0,C 180,E1 -3600.74,E2 -3600.74} C_VEL
LIN {X 0,Y 544.546,Z 756.728,A -85,B 0,C 180,E1 -3601.479,E2 -3601.479} C_VEL
LIN {X 0,Y 544.651,Z 754.392,A -85,B 0,C 180,E1 -3602.959,E2 -3602.959} C_VEL
LIN {X 0,Y 544.684,Z 751.514,A -85,B 0,C 180,E1 -3604.069,E2 -3604.069} C_VEL
LIN {X 0,Y 544.653,Z 747.599,A -85,B 0,C 180,E1 -3605.182,E2 -3605.182} C_VEL
LIN {X 0,Y 544.758,Z 743.417,A -85,B 0,C 180,E1 -3606.128,E2 -3606.128} C_VEL
LIN {X 0,Y 544.821,Z 737.363,A -85,B 0,C 180,E1 -3607.225,E2 -3607.225} C_VEL
LIN {X 0,Y 544.94,Z 731.129,A -85,B 0,C 180,E1 -3608.156,E2 -3608.156} C_VEL
LIN {X 0,Y 545.057,Z 723.622,A -85,B 0,C 180,E1 -3609.088,E2 -3609.088} C_VEL
LIN {X 0,Y 545.222,Z 716.519,A -85,B 0,C 180,E1 -3609.834,E2 -3609.834} C_VEL
LIN {X 0,Y 545.371,Z 708.077,A -85,B 0,C 180,E1 -3610.582,E2 -3610.582} C_VEL
LIN {X 0,Y 545.563,Z 698.57,A -85,B 0,C 180,E1 -3611.282,E2 -3611.282} C_VEL
LIN {X 0,Y 545.756,Z 688.454,A -85,B 0,C 180,E1 -3611.89,E2 -3611.89} C_VEL
LIN {X 0,Y 545.954,Z 675.395,A -85,B 0,C 180,E1 -3612.499,E2 -3612.499} C_VEL
LIN {X 0,Y 546.102,Z 663.267,A -85,B 0,C 180,E1 -3612.897,E2 -3612.897} C_VEL
LIN {X 0,Y 546.196,Z 652.943,A -85,B 0,C 180,E1 -3613.131,E2 -3613.131} C_VEL
LIN {X 0,Y 546.466,Z 551.261,A -85,B 0,C 180,E1 -3614.494,E2 -3614.494} C_VEL
LIN {X 0,Y 545.456,Z 544.736,A -85,B 0,C 180,E1 -3614.61,E2 -3614.61} C_VEL
LIN {X 0,Y 545.803,Z 523.539,A -85,B 0,C 180,E1 -3617.529,E2 -3617.529} C_VEL
LIN {X 0,Y 546.218,Z 502.041,A -85,B 0,C 180,E1 -3620.525,E2 -3620.525} C_VEL
LIN {X 0,Y 546.499,Z 479.7,A -85,B 0,C 180,E1 -3623.495,E2 -3623.495} C_VEL
LIN {X 0,Y 546.315,Z 473.784,A -85,B 0,C 180,E1 -3624.309,E2 -3624.309} C_VEL
LIN {X 0,Y 545.125,Z 467.71,A -85,B 0,C 180,E1 -3625.179,E2 -3625.179} C_VEL
LIN {X 0,Y 545.084,Z 467.71,A -85,B 0,C 180,E1 -3627.656,E2 -3627.656} C_VEL
LIN {X 0,Y 545.08,Z 467.712,A -85,B 0,C 180,E1 -3630.246,E2 -3630.246} C_VEL
LIN {X 0,Y 545.082,Z 467.713,A -85,B 0,C 180,E1 -3633.062,E2 -3633.062} C_VEL
LIN {X 0,Y 545.037,Z 467.714,A -85,B 0,C 180,E1 -3635.673,E2 -3635.673} C_VEL
LIN {X 0,Y 545.056,Z 467.715,A -85,B 0,C 180,E1 -3638.237,E2 -3638.237} C_VEL
LIN {X 0,Y 545.084,Z 467.715,A -85,B 0,C 180,E1 -3640.473,E2 -3640.473} C_VEL
LIN {X 0,Y 545.081,Z 467.709,A -85,B 0,C 180,E1 -3643.107,E2 -3643.107} C_VEL
LIN {X 0,Y 545.068,Z 467.714,A -85,B 0,C 180,E1 -3646.224,E2 -3646.224} C_VEL
LIN {X 0,Y 545.09,Z 467.71,A -85,B 0,C 180,E1 -3648.886,E2 -3648.886} C_VEL
LIN {X 0,Y 545.055,Z 467.712,A -85,B 0,C 180,E1 -3651.763,E2 -3651.763} C_VEL
LIN {X 0,Y 545.06,Z 467.718,A -85,B 0,C 180,E1 -3654.533,E2 -3654.533} C_VEL
LIN {X 0,Y 545.085,Z 467.708,A -85,B 0,C 180,E1 -3657.212,E2 -3657.212} C_VEL
LIN {X 0,Y 545.105,Z 467.708,A -85,B 0,C 180,E1 -3659.813,E2 -3659.813} C_VEL
LIN {X 0,Y 545.096,Z 467.711,A -85,B 0,C 180,E1 -3662.827,E2 -3662.827} C_VEL
LIN {X 0,Y 545.115,Z 467.808,A -85,B 0,C 180,E1 -3665.38,E2 -3665.38} C_VEL
LIN {X 0,Y 546.99,Z 476.177,A -85,B 0,C 180,E1 -3666.528,E2 -3666.528} C_VEL
LIN {X 0,Y 546.663,Z 493.736,A -85,B 0,C 180,E1 -3668.704,E2 -3668.704} C_VEL
LIN {X 0,Y 546.149,Z 519.293,A -85,B 0,C 180,E1 -3671.817,E2 -3671.817} C_VEL
LIN {X 0,Y 546.01,Z 523.721,A -85,B 0,C 180,E1 -3672.348,E2 -3672.348} C_VEL
LIN {X 0,Y 547.494,Z 533.872,A -85,B 0,C 180,E1 -3672.537,E2 -3672.537} C_VEL
LIN {X 0,Y 546.92,Z 662.882,A -85,B 0,C 180,E1 -3674.273,E2 -3674.273} C_VEL
LIN {X 0,Y 546.711,Z 677.376,A -85,B 0,C 180,E1 -3674.625,E2 -3674.625} C_VEL
LIN {X 0,Y 546.479,Z 691.834,A -85,B 0,C 180,E1 -3675.143,E2 -3675.143} C_VEL
LIN {X 0,Y 546.256,Z 704.638,A -85,B 0,C 180,E1 -3675.756,E2 -3675.756} C_VEL
LIN {X 0,Y 545.909,Z 717.1,A -85,B 0,C 180,E1 -3676.506,E2 -3676.506} C_VEL
LIN {X 0,Y 545.662,Z 729.646,A -85,B 0,C 180,E1 -3677.447,E2 -3677.447} C_VEL
LIN {X 0,Y 545.433,Z 740.838,A -85,B 0,C 180,E1 -3678.48,E2 -3678.48} C_VEL
LIN {X 0,Y 545.175,Z 750.852,A -85,B 0,C 180,E1 -3679.602,E2 -3679.602} C_VEL
LIN {X 0,Y 544.999,Z 759.174,A -85,B 0,C 180,E1 -3680.724,E2 -3680.724} C_VEL
LIN {X 0,Y 544.834,Z 767.127,A -85,B 0,C 180,E1 -3682.029,E2 -3682.029} C_VEL
LIN {X 0,Y 544.753,Z 773.876,A -85,B 0,C 180,E1 -3683.413,E2 -3683.413} C_VEL
LIN {X 0,Y 544.645,Z 779.201,A -85,B 0,C 180,E1 -3684.818,E2 -3684.818} C_VEL
LIN {X 0,Y 544.657,Z 783.316,A -85,B 0,C 180,E1 -3686.301,E2 -3686.301} C_VEL
LIN {X 0,Y 544.568,Z 786.002,A -85,B 0,C 180,E1 -3687.781,E2 -3687.781} C_VEL
LIN {X 0,Y 544.539,Z 787.333,A -85,B 0,C 180,E1 -3689.261,E2 -3689.261} C_VEL
LIN {X 0,Y 544.539,Z 787.334,A -85,B 0,C 180,E1 -3690.74,E2 -3690.74} C_VEL
LIN {X 0,Y 544.568,Z 786.004,A -85,B 0,C 180,E1 -3692.219,E2 -3692.219} C_VEL
LIN {X 0,Y 544.657,Z 783.319,A -85,B 0,C 180,E1 -3693.699,E2 -3693.699} C_VEL
LIN {X 0,Y 544.646,Z 779.201,A -85,B 0,C 180,E1 -3695.182,E2 -3695.182} C_VEL
LIN {X 0,Y 544.735,Z 773.948,A -85,B 0,C 180,E1 -3696.571,E2 -3696.571} C_VEL
LIN {X 0,Y 544.834,Z 767.127,A -85,B 0,C 180,E1 -3697.971,E2 -3697.971} C_VEL
LIN {X 0,Y 544.999,Z 759.174,A -85,B 0,C 180,E1 -3699.276,E2 -3699.276} C_VEL
LIN {X 0,Y 545.175,Z 750.852,A -85,B 0,C 180,E1 -3700.398,E2 -3700.398} C_VEL
LIN {X 0,Y 545.364,Z 741.027,A -85,B 0,C 180,E1 -3701.501,E2 -3701.501} C_VEL
LIN {X 0,Y 545.662,Z 729.644,A -85,B 0,C 180,E1 -3702.553,E2 -3702.553} C_VEL
LIN {X 0,Y 545.917,Z 717.101,A -85,B 0,C 180,E1 -3703.494,E2 -3703.494} C_VEL
LIN {X 0,Y 546.259,Z 704.637,A -85,B 0,C 180,E1 -3704.244,E2 -3704.244} C_VEL
LIN {X 0,Y 546.517,Z 690.693,A -85,B 0,C 180,E1 -3704.904,E2 -3704.904} C_VEL
LIN {X 0,Y 546.731,Z 676.553,A -85,B 0,C 180,E1 -3705.4,E2 -3705.4} C_VEL
LIN {X 0,Y 546.917,Z 662.875,A -85,B 0,C 180,E1 -3705.727,E2 -3705.727} C_VEL
LIN {X 0,Y 547.42,Z 532.217,A -85,B 0,C 180,E1 -3707.487,E2 -3707.487} C_VEL
LIN {X 0,Y 546.006,Z 523.738,A -85,B 0,C 180,E1 -3707.65,E2 -3707.65} C_VEL
LIN {X 0,Y 546.518,Z 498.479,A -85,B 0,C 180,E1 -3710.71,E2 -3710.71} C_VEL
LIN {X 0,Y 547.083,Z 477.835,A -85,B 0,C 180,E1 -3713.268,E2 -3713.268} C_VEL
LIN {X 0,Y 546.189,Z 472.408,A -85,B 0,C 180,E1 -3713.995,E2 -3713.995} C_VEL
LIN {X 0,Y 545.101,Z 467.711,A -85,B 0,C 180,E1 -3714.671,E2 -3714.671} C_VEL
LIN {X 0,Y 545.092,Z 467.715,A -85,B 0,C 180,E1 -3717.656,E2 -3717.656} C_VEL
LIN {X 0,Y 545.08,Z 467.712,A -85,B 0,C 180,E1 -3720.246,E2 -3720.246} C_VEL
LIN {X 0,Y 545.083,Z 467.713,A -85,B 0,C 180,E1 -3723.063,E2 -3723.063} C_VEL
LIN {X 0,Y 545.036,Z 467.72,A -85,B 0,C 180,E1 -3725.673,E2 -3725.673} C_VEL
LIN {X 0,Y 545.055,Z 467.712,A -85,B 0,C 180,E1 -3728.237,E2 -3728.237} C_VEL
LIN {X 0,Y 545.086,Z 467.715,A -85,B 0,C 180,E1 -3731.115,E2 -3731.115} C_VEL
LIN {X 0,Y 545.061,Z 467.711,A -85,B 0,C 180,E1 -3734.129,E2 -3734.129} C_VEL
LIN {X 0,Y 545.065,Z 467.716,A -85,B 0,C 180,E1 -3737.303,E2 -3737.303} C_VEL
LIN {X 0,Y 545.075,Z 467.71,A -85,B 0,C 180,E1 -3739.858,E2 -3739.858} C_VEL
LIN {X 0,Y 545.074,Z 467.716,A -85,B 0,C 180,E1 -3743.074,E2 -3743.074} C_VEL
LIN {X 0,Y 545.074,Z 467.713,A -85,B 0,C 180,E1 -3746.329,E2 -3746.329} C_VEL
LIN {X 0,Y 545.072,Z 467.717,A -85,B 0,C 180,E1 -3748.952,E2 -3748.952} C_VEL
LIN {X 0,Y 545.107,Z 467.71,A -85,B 0,C 180,E1 -3751.508,E2 -3751.508} C_VEL
LIN {X 0,Y 545.1,Z 467.716,A -85,B 0,C 180,E1 -3754.491,E2 -3754.491} C_VEL
LIN {X 0,Y 545.117,Z 467.907,A -85,B 0,C 180,E1 -3755.879,E2 -3755.879} C_VEL
LIN {X 0,Y 546.679,Z 475.826,A -85,B 0,C 180,E1 -3757.115,E2 -3757.115} C_VEL
LIN {X 0,Y 546.261,Z 495.25,A -85,B 0,C 180,E1 -3759.917,E2 -3759.917} C_VEL
LIN {X 0,Y 545.854,Z 516.771,A -85,B 0,C 180,E1 -3762.968,E2 -3762.968} C_VEL
LIN {X 0,Y 545.469,Z 538.534,A -85,B 0,C 180,E1 -3766.02,E2 -3766.02} C_VEL
LIN {X 0,Y 545.403,Z 541.854,A -85,B 0,C 180,E1 -3766.482,E2 -3766.482} C_VEL
LIN {X 0,Y 546.546,Z 549.692,A -85,B 0,C 180,E1 -3766.617,E2 -3766.617} C_VEL
LIN {X 0,Y 546.205,Z 650.804,A -85,B 0,C 180,E1 -3767.969,E2 -3767.969} C_VEL
LIN {X 0,Y 546.071,Z 663.983,A -85,B 0,C 180,E1 -3768.299,E2 -3768.299} C_VEL
LIN {X 0,Y 545.879,Z 676.751,A -85,B 0,C 180,E1 -3768.774,E2 -3768.774} C_VEL
LIN {X 0,Y 545.759,Z 687.947,A -85,B 0,C 180,E1 -3769.332,E2 -3769.332} C_VEL
LIN {X 0,Y 545.455,Z 699.508,A -85,B 0,C 180,E1 -3770.077,E2 -3770.077} C_VEL
LIN {X 0,Y 545.286,Z 709.897,A -85,B 0,C 180,E1 -3770.916,E2 -3770.916} C_VEL
LIN {X 0,Y 545.089,Z 719.303,A -85,B 0,C 180,E1 -3771.846,E2 -3771.846} C_VEL
LIN {X 0,Y 544.939,Z 727.129,A -85,B 0,C 180,E1 -3772.795,E2 -3772.795} C_VEL
LIN {X 0,Y 544.892,Z 734.069,A -85,B 0,C 180,E1 -3773.815,E2 -3773.815} C_VEL
LIN {X 0,Y 544.681,Z 739.702,A -85,B 0,C 180,E1 -3774.818,E2 -3774.818} C_VEL
LIN {X 0,Y 544.706,Z 744.689,A -85,B 0,C 180,E1 -3775.931,E2 -3775.931} C_VEL
LIN {X 0,Y 544.672,Z 748.589,A -85,B 0,C 180,E1 -3777.041,E2 -3777.041} C_VEL
LIN {X 0,Y 544.591,Z 750.597,A -85,B 0,C 180,E1 -3777.781,E2 -3777.781} C_VEL
LIN {X 0,Y 544.551,Z 752.166,A -85,B 0,C 180,E1 -3778.521,E2 -3778.521} C_VEL
LIN {X 0,Y 544.543,Z 753.322,A -85,B 0,C 180,E1 -3779.26,E2 -3779.26} C_VEL
LIN {X 0,Y 544.542,Z 754.079,A -85,B 0,C 180,E1 -3780,E2 -3780} C_VEL
LIN {X 0,Y 544.545,Z 754.397,A -85,B 0,C 180,E1 -3781.479,E2 -3781.479} C_VEL
LIN {X 0,Y 544.569,Z 753.968,A -85,B 0,C 180,E1 -3782.219,E2 -3782.219} C_VEL
LIN {X 0,Y 544.646,Z 753.136,A -85,B 0,C 180,E1 -3782.959,E2 -3782.959} C_VEL
LIN {X 0,Y 544.653,Z 751.901,A -85,B 0,C 180,E1 -3783.699,E2 -3783.699} C_VEL
LIN {X 0,Y 544.602,Z 749.283,A -85,B 0,C 180,E1 -3784.812,E2 -3784.812} C_VEL
LIN {X 0,Y 544.704,Z 745.595,A -85,B 0,C 180,E1 -3785.925,E2 -3785.925} C_VEL
LIN {X 0,Y 544.734,Z 740.856,A -85,B 0,C 180,E1 -3787.04,E2 -3787.04} C_VEL
LIN {X 0,Y 544.832,Z 734.783,A -85,B 0,C 180,E1 -3788.157,E2 -3788.157} C_VEL
LIN {X 0,Y 544.963,Z 727.26,A -85,B 0,C 180,E1 -3789.277,E2 -3789.277} C_VEL
LIN {X 0,Y 545.088,Z 719.595,A -85,B 0,C 180,E1 -3790.212,E2 -3790.212} C_VEL
LIN {X 0,Y 545.284,Z 710.202,A -85,B 0,C 180,E1 -3791.147,E2 -3791.147} C_VEL
LIN {X 0,Y 545.482,Z 699.802,A -85,B 0,C 180,E1 -3791.991,E2 -3791.991} C_VEL
LIN {X 0,Y 545.707,Z 688.249,A -85,B 0,C 180,E1 -3792.741,E2 -3792.741} C_VEL
LIN {X 0,Y 545.893,Z 675.975,A -85,B 0,C 180,E1 -3793.352,E2 -3793.352} C_VEL
LIN {X 0,Y 546.033,Z 663.75,A -85,B 0,C 180,E1 -3793.799,E2 -3793.799} C_VEL
LIN {X 0,Y 546.216,Z 651.8,A -85,B 0,C 180,E1 -3794.103,E2 -3794.103} C_VEL
LIN {X 0,Y 546.383,Z 607.014,A -85,B 0,C 180,E1 -3794.717,E2 -3794.717} C_VEL
LIN {X 0,Y 546.457,Z 548.599,A -85,B 0,C 180,E1 -3795.49,E2 -3795.49} C_VEL
LIN {X 0,Y 545.417,Z 541.744,A -85,B 0,C 180,E1 -3795.623,E2 -3795.623} C_VEL
LIN {X 0,Y 545.792,Z 520.576,A -85,B 0,C 180,E1 -3798.584,E2 -3798.584} C_VEL
LIN {X 0,Y 546.142,Z 501.474,A -85,B 0,C 180,E1 -3801.292,E2 -3801.292} C_VEL
LIN {X 0,Y 545.58,Z 498.11,A -85,B 0,C 180,E1 -3801.798,E2 -3801.798} C_VEL
LIN {X 0,Y 540.22,Z 487.911,A -85,B 0,C 180,E1 -3803.507,E2 -3803.507} C_VEL
LIN {X 0,Y 539.681,Z 484.565,A -85,B 0,C 180,E1 -3804.023,E2 -3804.023} C_VEL
LIN {X 0,Y 539.68,Z 476.309,A -85,B 0,C 180,E1 -3805.245,E2 -3805.245} C_VEL
LIN {X 0,Y 538.076,Z 468.586,A -85,B 0,C 180,E1 -3806.495,E2 -3806.495} C_VEL
LIN {X 0,Y 538.034,Z 468.589,A -85,B 0,C 180,E1 -3808.933,E2 -3808.933} C_VEL
LIN {X 0,Y 538.013,Z 468.594,A -85,B 0,C 180,E1 -3811.887,E2 -3811.887} C_VEL
LIN {X 0,Y 538.031,Z 468.586,A -85,B 0,C 180,E1 -3814.62,E2 -3814.62} C_VEL
LIN {X 0,Y 538.009,Z 468.591,A -85,B 0,C 180,E1 -3817.17,E2 -3817.17} C_VEL
LIN {X 0,Y 538.028,Z 468.592,A -85,B 0,C 180,E1 -3819.797,E2 -3819.797} C_VEL
LIN {X 0,Y 538.021,Z 468.586,A -85,B 0,C 180,E1 -3822.786,E2 -3822.786} C_VEL
LIN {X 0,Y 538.033,Z 468.589,A -85,B 0,C 180,E1 -3825.925,E2 -3825.925} C_VEL
LIN {X 0,Y 538.051,Z 468.587,A -85,B 0,C 180,E1 -3829.253,E2 -3829.253} C_VEL
LIN {X 0,Y 537.995,Z 468.591,A -85,B 0,C 180,E1 -3832.122,E2 -3832.122} C_VEL
LIN {X 0,Y 538,Z 468.59,A -85,B 0,C 180,E1 -3834.915,E2 -3834.915} C_VEL
LIN {X 0,Y 538.021,Z 468.595,A -85,B 0,C 180,E1 -3837.617,E2 -3837.617} C_VEL
LIN {X 0,Y 538.019,Z 468.587,A -85,B 0,C 180,E1 -3840.239,E2 -3840.239} C_VEL
LIN {X 0,Y 538.06,Z 468.582,A -85,B 0,C 180,E1 -3842.796,E2 -3842.796} C_VEL
LIN {X 0,Y 538.05,Z 468.588,A -85,B 0,C 180,E1 -3845.292,E2 -3845.292} C_VEL
LIN {X 0,Y 538.025,Z 468.586,A -85,B 0,C 180,E1 -3848.546,E2 -3848.546} C_VEL
LIN {X 0,Y 538.04,Z 468.586,A -85,B 0,C 180,E1 -3850.94,E2 -3850.94} C_VEL
LIN {X 0,Y 538.028,Z 468.592,A -85,B 0,C 180,E1 -3853.299,E2 -3853.299} C_VEL
LIN {X 0,Y 538.067,Z 468.588,A -85,B 0,C 180,E1 -3855.631,E2 -3855.631} C_VEL
LIN {X 0,Y 538.08,Z 468.579,A -85,B 0,C 180,E1 -3858.701,E2 -3858.701} C_VEL
LIN {X 0,Y 538.093,Z 468.583,A -85,B 0,C 180,E1 -3861.74,E2 -3861.74} C_VEL
LIN {X 0,Y 538.165,Z 468.569,A -85,B 0,C 180,E1 -3864.755,E2 -3864.755} C_VEL
LIN {X 0,Y 538.172,Z 468.572,A -85,B 0,C 180,E1 -3867.755,E2 -3867.755} C_VEL
LIN {X 0,Y 538.184,Z 468.567,A -85,B 0,C 180,E1 -3870.748,E2 -3870.748} C_VEL
LIN {X 0,Y 538.141,Z 468.574,A -85,B 0,C 180,E1 -3872.994,E2 -3872.994} C_VEL
LIN {X 0,Y 538.124,Z 468.575,A -85,B 0,C 180,E1 -3875.997,E2 -3875.997} C_VEL
LIN {X 0,Y 538.071,Z 468.583,A -85,B 0,C 180,E1 -3879.018,E2 -3879.018} C_VEL
LIN {X 0,Y 538.086,Z 468.579,A -85,B 0,C 180,E1 -3882.062,E2 -3882.062} C_VEL
LIN {X 0,Y 538.048,Z 468.588,A -85,B 0,C 180,E1 -3885.144,E2 -3885.144} C_VEL
LIN {X 0,Y 538.032,Z 468.585,A -85,B 0,C 180,E1 -3888.27,E2 -3888.27} C_VEL
LIN {X 0,Y 538.042,Z 468.584,A -85,B 0,C 180,E1 -3890.651,E2 -3890.651} C_VEL
LIN {X 0,Y 538.027,Z 468.588,A -85,B 0,C 180,E1 -3893.887,E2 -3893.887} C_VEL
LIN {X 0,Y 538.044,Z 468.583,A -85,B 0,C 180,E1 -3896.367,E2 -3896.367} C_VEL
LIN {X 0,Y 538.033,Z 468.588,A -85,B 0,C 180,E1 -3898.934,E2 -3898.934} C_VEL
LIN {X 0,Y 538.013,Z 468.589,A -85,B 0,C 180,E1 -3901.887,E2 -3901.887} C_VEL
LIN {X 0,Y 538.014,Z 468.588,A -85,B 0,C 180,E1 -3904.618,E2 -3904.618} C_VEL
LIN {X 0,Y 538.007,Z 468.595,A -85,B 0,C 180,E1 -3907.17,E2 -3907.17} C_VEL
LIN {X 0,Y 538.029,Z 468.588,A -85,B 0,C 180,E1 -3909.797,E2 -3909.797} C_VEL
LIN {X 0,Y 538.026,Z 468.588,A -85,B 0,C 180,E1 -3912.786,E2 -3912.786} C_VEL
LIN {X 0,Y 538.032,Z 468.592,A -85,B 0,C 180,E1 -3915.14,E2 -3915.14} C_VEL
LIN {X 0,Y 538.032,Z 468.585,A -85,B 0,C 180,E1 -3918.227,E2 -3918.227} C_VEL
LIN {X 0,Y 538.017,Z 468.594,A -85,B 0,C 180,E1 -3921.17,E2 -3921.17} C_VEL
LIN {X 0,Y 537.997,Z 468.589,A -85,B 0,C 180,E1 -3924.089,E2 -3924.089} C_VEL
LIN {X 0,Y 538.033,Z 468.587,A -85,B 0,C 180,E1 -3926.728,E2 -3926.728} C_VEL
LIN {X 0,Y 538.029,Z 468.591,A -85,B 0,C 180,E1 -3929.556,E2 -3929.556} C_VEL
LIN {X 0,Y 538.043,Z 468.586,A -85,B 0,C 180,E1 -3931.95,E2 -3931.95} C_VEL
LIN {X 0,Y 538.108,Z 468.675,A -85,B 0,C 180,E1 -3934.599,E2 -3934.599} C_VEL
LIN {X 0,Y 539.714,Z 477.241,A -85,B 0,C 180,E1 -3935.861,E2 -3935.861} C_VEL
LIN {X 0,Y 539.429,Z 494.049,A -85,B 0,C 180,E1 -3938.203,E2 -3938.203} C_VEL
LIN {X 0,Y 538.991,Z 515.092,A -85,B 0,C 180,E1 -3941.173,E2 -3941.173} C_VEL
LIN {X 0,Y 538.639,Z 534.826,A -85,B 0,C 180,E1 -3943.903,E2 -3943.903} C_VEL
LIN {X 0,Y 538.487,Z 544.865,A -85,B 0,C 180,E1 -3945.291,E2 -3945.291} C_VEL
LIN {X 0,Y 539.676,Z 553.566,A -85,B 0,C 180,E1 -3945.441,E2 -3945.441} C_VEL
LIN {X 0,Y 539.343,Z 651.857,A -85,B 0,C 180,E1 -3946.771,E2 -3946.771} C_VEL
LIN {X 0,Y 539.194,Z 662.551,A -85,B 0,C 180,E1 -3947.006,E2 -3947.006} C_VEL
LIN {X 0,Y 539.045,Z 672.903,A -85,B 0,C 180,E1 -3947.338,E2 -3947.338} C_VEL
LIN {X 0,Y 538.876,Z 685.017,A -85,B 0,C 180,E1 -3947.86,E2 -3947.86} C_VEL
LIN {X 0,Y 538.67,Z 695.566,A -85,B 0,C 180,E1 -3948.458,E2 -3948.458} C_VEL
LIN {X 0,Y 538.428,Z 705.785,A -85,B 0,C 180,E1 -3949.185,E2 -3949.185} C_VEL
LIN {X 0,Y 538.245,Z 713.578,A -85,B 0,C 180,E1 -3949.847,E2 -3949.847} C_VEL
LIN {X 0,Y 538.086,Z 721.125,A -85,B 0,C 180,E1 -3950.604,E2 -3950.604} C_VEL
LIN {X 0,Y 537.974,Z 727.605,A -85,B 0,C 180,E1 -3951.36,E2 -3951.36} C_VEL
LIN {X 0,Y 537.82,Z 734.411,A -85,B 0,C 180,E1 -3952.303,E2 -3952.303} C_VEL
LIN {X 0,Y 537.698,Z 740.886,A -85,B 0,C 180,E1 -3953.396,E2 -3953.396} C_VEL
LIN {X 0,Y 537.675,Z 745.623,A -85,B 0,C 180,E1 -3954.374,E2 -3954.374} C_VEL
LIN {X 0,Y 537.562,Z 749.971,A -85,B 0,C 180,E1 -3955.501,E2 -3955.501} C_VEL
LIN {X 0,Y 537.591,Z 752.343,A -85,B 0,C 180,E1 -3956.252,E2 -3956.252} C_VEL
LIN {X 0,Y 537.551,Z 754.177,A -85,B 0,C 180,E1 -3957.002,E2 -3957.002} C_VEL
LIN {X 0,Y 537.452,Z 756.644,A -85,B 0,C 180,E1 -3958.501,E2 -3958.501} C_VEL
LIN {X 0,Y 537.442,Z 757.246,A -85,B 0,C 180,E1 -3959.251,E2 -3959.251} C_VEL
LIN {X 0,Y 537.442,Z 757.309,A -85,B 0,C 180,E1 -3960.749,E2 -3960.749} C_VEL
LIN {X 0,Y 537.451,Z 756.72,A -85,B 0,C 180,E1 -3961.499,E2 -3961.499} C_VEL
LIN {X 0,Y 537.552,Z 754.388,A -85,B 0,C 180,E1 -3962.998,E2 -3962.998} C_VEL
LIN {X 0,Y 537.603,Z 751.507,A -85,B 0,C 180,E1 -3964.123,E2 -3964.123} C_VEL
LIN {X 0,Y 537.587,Z 747.59,A -85,B 0,C 180,E1 -3965.251,E2 -3965.251} C_VEL
LIN {X 0,Y 537.637,Z 742.843,A -85,B 0,C 180,E1 -3966.319,E2 -3966.319} C_VEL
LIN {X 0,Y 537.753,Z 737.35,A -85,B 0,C 180,E1 -3967.321,E2 -3967.321} C_VEL
LIN {X 0,Y 537.886,Z 731.115,A -85,B 0,C 180,E1 -3968.264,E2 -3968.264} C_VEL
LIN {X 0,Y 538.021,Z 723.607,A -85,B 0,C 180,E1 -3969.208,E2 -3969.208} C_VEL
LIN {X 0,Y 538.216,Z 716.503,A -85,B 0,C 180,E1 -3969.963,E2 -3969.963} C_VEL
LIN {X 0,Y 538.369,Z 708.061,A -85,B 0,C 180,E1 -3970.721,E2 -3970.721} C_VEL
LIN {X 0,Y 538.547,Z 700.619,A -85,B 0,C 180,E1 -3971.289,E2 -3971.289} C_VEL
LIN {X 0,Y 538.742,Z 691.552,A -85,B 0,C 180,E1 -3971.869,E2 -3971.869} C_VEL
LIN {X 0,Y 538.873,Z 681.813,A -85,B 0,C 180,E1 -3972.379,E2 -3972.379} C_VEL
LIN {X 0,Y 539.06,Z 671.431,A -85,B 0,C 180,E1 -3972.805,E2 -3972.805} C_VEL
LIN {X 0,Y 539.222,Z 660.558,A -85,B 0,C 180,E1 -3973.137,E2 -3973.137} C_VEL
LIN {X 0,Y 539.365,Z 647.373,A -85,B 0,C 180,E1 -3973.397,E2 -3973.397} C_VEL
LIN {X 0,Y 539.567,Z 551.722,A -85,B 0,C 180,E1 -3974.677,E2 -3974.677} C_VEL
LIN {X 0,Y 538.493,Z 544.594,A -85,B 0,C 180,E1 -3974.823,E2 -3974.823} C_VEL
LIN {X 0,Y 538.857,Z 522.149,A -85,B 0,C 180,E1 -3977.951,E2 -3977.951} C_VEL
LIN {X 0,Y 539.252,Z 503.126,A -85,B 0,C 180,E1 -3980.603,E2 -3980.603} C_VEL
LIN {X 0,Y 539.549,Z 480.69,A -85,B 0,C 180,E1 -3983.612,E2 -3983.612} C_VEL
LIN {X 0,Y 539.344,Z 475.002,A -85,B 0,C 180,E1 -3984.385,E2 -3984.385} C_VEL
LIN {X 0,Y 538.079,Z 468.587,A -85,B 0,C 180,E1 -3985.274,E2 -3985.274} C_VEL
LIN {X 0,Y 538.043,Z 468.588,A -85,B 0,C 180,E1 -3988.05,E2 -3988.05} C_VEL
LIN {X 0,Y 538.023,Z 468.596,A -85,B 0,C 180,E1 -3990.627,E2 -3990.627} C_VEL
LIN {X 0,Y 538.048,Z 468.587,A -85,B 0,C 180,E1 -3993.283,E2 -3993.283} C_VEL
LIN {X 0,Y 537.997,Z 468.592,A -85,B 0,C 180,E1 -3996.004,E2 -3996.004} C_VEL
LIN {X 0,Y 538.018,Z 468.594,A -85,B 0,C 180,E1 -3998.83,E2 -3998.83} C_VEL
LIN {X 0,Y 538.032,Z 468.586,A -85,B 0,C 180,E1 -4001.773,E2 -4001.773} C_VEL
LIN {X 0,Y 538.034,Z 468.59,A -85,B 0,C 180,E1 -4004.859,E2 -4004.859} C_VEL
LIN {X 0,Y 538.038,Z 468.589,A -85,B 0,C 180,E1 -4008.121,E2 -4008.121} C_VEL
LIN {X 0,Y 538.015,Z 468.589,A -85,B 0,C 180,E1 -4011.17,E2 -4011.17} C_VEL
LIN {X 0,Y 538.03,Z 468.591,A -85,B 0,C 180,E1 -4014.084,E2 -4014.084} C_VEL
LIN {X 0,Y 538.034,Z 468.59,A -85,B 0,C 180,E1 -4016.727,E2 -4016.727} C_VEL
LIN {X 0,Y 538.041,Z 468.586,A -85,B 0,C 180,E1 -4019.554,E2 -4019.554} C_VEL
LIN {X 0,Y 538.047,Z 468.59,A -85,B 0,C 180,E1 -4021.95,E2 -4021.95} C_VEL
LIN {X 0,Y 538.085,Z 468.641,A -85,B 0,C 180,E1 -4025.14,E2 -4025.14} C_VEL
LIN {X 0,Y 540.144,Z 477.806,A -85,B 0,C 180,E1 -4026.416,E2 -4026.416} C_VEL
LIN {X 0,Y 539.773,Z 495.365,A -85,B 0,C 180,E1 -4028.619,E2 -4028.619} C_VEL
LIN {X 0,Y 539.207,Z 520.912,A -85,B 0,C 180,E1 -4031.771,E2 -4031.771} C_VEL
LIN {X 0,Y 539.115,Z 523.791,A -85,B 0,C 180,E1 -4032.122,E2 -4032.122} C_VEL
LIN {X 0,Y 540.717,Z 534.321,A -85,B 0,C 180,E1 -4032.32,E2 -4032.32} C_VEL
LIN {X 0,Y 540.089,Z 662.882,A -85,B 0,C 180,E1 -4034.069,E2 -4034.069} C_VEL
LIN {X 0,Y 539.861,Z 677.486,A -85,B 0,C 180,E1 -4034.428,E2 -4034.428} C_VEL
LIN {X 0,Y 539.623,Z 691.833,A -85,B 0,C 180,E1 -4034.95,E2 -4034.95} C_VEL
LIN {X 0,Y 539.37,Z 704.636,A -85,B 0,C 180,E1 -4035.57,E2 -4035.57} C_VEL
LIN {X 0,Y 538.996,Z 717.098,A -85,B 0,C 180,E1 -4036.33,E2 -4036.33} C_VEL
LIN {X 0,Y 538.684,Z 729.648,A -85,B 0,C 180,E1 -4037.281,E2 -4037.281} C_VEL
LIN {X 0,Y 538.434,Z 739.821,A -85,B 0,C 180,E1 -4038.223,E2 -4038.223} C_VEL
LIN {X 0,Y 538.204,Z 749.333,A -85,B 0,C 180,E1 -4039.276,E2 -4039.276} C_VEL
LIN {X 0,Y 537.968,Z 757.91,A -85,B 0,C 180,E1 -4040.412,E2 -4040.412} C_VEL
LIN {X 0,Y 537.805,Z 766.118,A -85,B 0,C 180,E1 -4041.735,E2 -4041.735} C_VEL
LIN {X 0,Y 537.661,Z 771.863,A -85,B 0,C 180,E1 -4042.867,E2 -4042.867} C_VEL
LIN {X 0,Y 537.654,Z 777.961,A -85,B 0,C 180,E1 -4044.374,E2 -4044.374} C_VEL
LIN {X 0,Y 537.55,Z 781.444,A -85,B 0,C 180,E1 -4045.501,E2 -4045.501} C_VEL
LIN {X 0,Y 537.547,Z 784.832,A -85,B 0,C 180,E1 -4047.002,E2 -4047.002} C_VEL
LIN {X 0,Y 537.446,Z 786.834,A -85,B 0,C 180,E1 -4048.501,E2 -4048.501} C_VEL
LIN {X 0,Y 537.44,Z 787.5,A -85,B 0,C 180,E1 -4050,E2 -4050} C_VEL
LIN {X 0,Y 537.446,Z 786.835,A -85,B 0,C 180,E1 -4051.499,E2 -4051.499} C_VEL
LIN {X 0,Y 537.547,Z 784.835,A -85,B 0,C 180,E1 -4052.998,E2 -4052.998} C_VEL
LIN {X 0,Y 537.55,Z 781.447,A -85,B 0,C 180,E1 -4054.499,E2 -4054.499} C_VEL
LIN {X 0,Y 537.647,Z 776.567,A -85,B 0,C 180,E1 -4056.003,E2 -4056.003} C_VEL
LIN {X 0,Y 537.704,Z 770.054,A -85,B 0,C 180,E1 -4057.51,E2 -4057.51} C_VEL
LIN {X 0,Y 537.86,Z 762.803,A -85,B 0,C 180,E1 -4058.832,E2 -4058.832} C_VEL
LIN {X 0,Y 538.048,Z 753.821,A -85,B 0,C 180,E1 -4060.157,E2 -4060.157} C_VEL
LIN {X 0,Y 538.319,Z 744.391,A -85,B 0,C 180,E1 -4061.293,E2 -4061.293} C_VEL
LIN {X 0,Y 538.565,Z 733.951,A -85,B 0,C 180,E1 -4062.339,E2 -4062.339} C_VEL
LIN {X 0,Y 538.881,Z 722.426,A -85,B 0,C 180,E1 -4063.289,E2 -4063.289} C_VEL
LIN {X 0,Y 539.208,Z 709.636,A -85,B 0,C 180,E1 -4064.146,E2 -4064.146} C_VEL
LIN {X 0,Y 539.503,Z 697.142,A -85,B 0,C 180,E1 -4064.812,E2 -4064.812} C_VEL
LIN {X 0,Y 539.795,Z 683.829,A -85,B 0,C 180,E1 -4065.362,E2 -4065.362} C_VEL
LIN {X 0,Y 540.011,Z 669.774,A -85,B 0,C 180,E1 -4065.782,E2 -4065.782} C_VEL
LIN {X 0,Y 540.168,Z 655.591,A -85,B 0,C 180,E1 -4066.05,E2 -4066.05} C_VEL
LIN {X 0,Y 540.65,Z 532.865,A -85,B 0,C 180,E1 -4067.701,E2 -4067.701} C_VEL
LIN {X 0,Y 539.098,Z 523.706,A -85,B 0,C 180,E1 -4067.886,E2 -4067.886} C_VEL
LIN {X 0,Y 539.682,Z 498.462,A -85,B 0,C 180,E1 -4070.985,E2 -4070.985} C_VEL
LIN {X 0,Y 540.26,Z 479.487,A -85,B 0,C 180,E1 -4073.376,E2 -4073.376} C_VEL
LIN {X 0,Y 539.247,Z 473.638,A -85,B 0,C 180,E1 -4074.173,E2 -4074.173} C_VEL
LIN {X 0,Y 538.077,Z 468.587,A -85,B 0,C 180,E1 -4074.912,E2 -4074.912} C_VEL
LIN {X 0,Y 538.047,Z 468.591,A -85,B 0,C 180,E1 -4078.05,E2 -4078.05} C_VEL
LIN {X 0,Y 538.024,Z 468.59,A -85,B 0,C 180,E1 -4080.627,E2 -4080.627} C_VEL
LIN {X 0,Y 538.048,Z 468.592,A -85,B 0,C 180,E1 -4083.283,E2 -4083.283} C_VEL
LIN {X 0,Y 537.997,Z 468.593,A -85,B 0,C 180,E1 -4086.005,E2 -4086.005} C_VEL
LIN {X 0,Y 538.016,Z 468.592,A -85,B 0,C 180,E1 -4088.831,E2 -4088.831} C_VEL
LIN {X 0,Y 538.035,Z 468.588,A -85,B 0,C 180,E1 -4091.773,E2 -4091.773} C_VEL
LIN {X 0,Y 538.033,Z 468.592,A -85,B 0,C 180,E1 -4094.86,E2 -4094.86} C_VEL
LIN {X 0,Y 538.035,Z 468.586,A -85,B 0,C 180,E1 -4098.121,E2 -4098.121} C_VEL
LIN {X 0,Y 538.041,Z 468.588,A -85,B 0,C 180,E1 -4100.415,E2 -4100.415} C_VEL
LIN {X 0,Y 538.028,Z 468.594,A -85,B 0,C 180,E1 -4103.067,E2 -4103.067} C_VEL
LIN {X 0,Y 538.029,Z 468.588,A -85,B 0,C 180,E1 -4105.827,E2 -4105.827} C_VEL
LIN {X 0,Y 538.015,Z 468.595,A -85,B 0,C 180,E1 -4108.499,E2 -4108.499} C_VEL
LIN {X 0,Y 538.064,Z 468.59,A -85,B 0,C 180,E1 -4111.1,E2 -4111.1} C_VEL
LIN {X 0,Y 538.047,Z 468.591,A -85,B 0,C 180,E1 -4113.634,E2 -4113.634} C_VEL
LIN {X 0,Y 538.049,Z 468.722,A -85,B 0,C 180,E1 -4115.653,E2 -4115.653} C_VEL
LIN {X 0,Y 539.801,Z 477.257,A -85,B 0,C 180,E1 -4117.009,E2 -4117.009} C_VEL
LIN {X 0,Y 539.345,Z 496.049,A -85,B 0,C 180,E1 -4119.753,E2 -4119.753} C_VEL
LIN {X 0,Y 538.912,Z 516.874,A -85,B 0,C 180,E1 -4122.741,E2 -4122.741} C_VEL
LIN {X 0,Y 538.494,Z 538.642,A -85,B 0,C 180,E1 -4125.835,E2 -4125.835} C_VEL
LIN {X 0,Y 538.448,Z 541.702,A -85,B 0,C 180,E1 -4126.267,E2 -4126.267} C_VEL
LIN {X 0,Y 539.697,Z 550.738,A -85,B 0,C 180,E1 -4126.444,E2 -4126.444} C_VEL
LIN {X 0,Y 539.296,Z 650.484,A -85,B 0,C 180,E1 -4127.793,E2 -4127.793} C_VEL
LIN {X 0,Y 539.188,Z 663.468,A -85,B 0,C 180,E1 -4128.118,E2 -4128.118} C_VEL
LIN {X 0,Y 538.982,Z 675.196,A -85,B 0,C 180,E1 -4128.543,E2 -4128.543} C_VEL
LIN {X 0,Y 538.83,Z 686.453,A -85,B 0,C 180,E1 -4129.098,E2 -4129.098} C_VEL
LIN {X 0,Y 538.584,Z 697.049,A -85,B 0,C 180,E1 -4129.759,E2 -4129.759} C_VEL
LIN {X 0,Y 538.342,Z 706.883,A -85,B 0,C 180,E1 -4130.513,E2 -4130.513} C_VEL
LIN {X 0,Y 538.176,Z 715.877,A -85,B 0,C 180,E1 -4131.363,E2 -4131.363} C_VEL
LIN {X 0,Y 537.949,Z 724.212,A -85,B 0,C 180,E1 -4132.304,E2 -4132.304} C_VEL
LIN {X 0,Y 537.79,Z 731.505,A -85,B 0,C 180,E1 -4133.313,E2 -4133.313} C_VEL
LIN {X 0,Y 537.712,Z 737.82,A -85,B 0,C 180,E1 -4134.374,E2 -4134.374} C_VEL
LIN {X 0,Y 537.638,Z 743.235,A -85,B 0,C 180,E1 -4135.502,E2 -4135.502} C_VEL
LIN {X 0,Y 537.636,Z 747.434,A -85,B 0,C 180,E1 -4136.628,E2 -4136.628} C_VEL
LIN {X 0,Y 537.51,Z 750.629,A -85,B 0,C 180,E1 -4137.752,E2 -4137.752} C_VEL
LIN {X 0,Y 537.456,Z 752.191,A -85,B 0,C 180,E1 -4138.501,E2 -4138.501} C_VEL
LIN {X 0,Y 537.443,Z 753.339,A -85,B 0,C 180,E1 -4139.251,E2 -4139.251} C_VEL
LIN {X 0,Y 537.443,Z 754.087,A -85,B 0,C 180,E1 -4140,E2 -4140} C_VEL
LIN {X 0,Y 537.451,Z 754.39,A -85,B 0,C 180,E1 -4141.499,E2 -4141.499} C_VEL
LIN {X 0,Y 537.488,Z 753.953,A -85,B 0,C 180,E1 -4142.248,E2 -4142.248} C_VEL
LIN {X 0,Y 537.546,Z 753.114,A -85,B 0,C 180,E1 -4142.998,E2 -4142.998} C_VEL
LIN {X 0,Y 537.57,Z 751.87,A -85,B 0,C 180,E1 -4143.748,E2 -4143.748} C_VEL
LIN {X 0,Y 537.517,Z 749.245,A -85,B 0,C 180,E1 -4144.875,E2 -4144.875} C_VEL
LIN {X 0,Y 537.613,Z 745.54,A -85,B 0,C 180,E1 -4146.003,E2 -4146.003} C_VEL
LIN {X 0,Y 537.655,Z 740.791,A -85,B 0,C 180,E1 -4147.133,E2 -4147.133} C_VEL
LIN {X 0,Y 537.757,Z 734.698,A -85,B 0,C 180,E1 -4148.265,E2 -4148.265} C_VEL
LIN {X 0,Y 537.908,Z 727.15,A -85,B 0,C 180,E1 -4149.4,E2 -4149.4} C_VEL
LIN {X 0,Y 538.072,Z 719.474,A -85,B 0,C 180,E1 -4150.346,E2 -4150.346} C_VEL
LIN {X 0,Y 538.26,Z 710.045,A -85,B 0,C 180,E1 -4151.295,E2 -4151.295} C_VEL
LIN {X 0,Y 538.507,Z 699.601,A -85,B 0,C 180,E1 -4152.148,E2 -4152.148} C_VEL
LIN {X 0,Y 538.722,Z 689.62,A -85,B 0,C 180,E1 -4152.813,E2 -4152.813} C_VEL
LIN {X 0,Y 538.899,Z 677.725,A -85,B 0,C 180,E1 -4153.433,E2 -4153.433} C_VEL
LIN {X 0,Y 539.092,Z 664.828,A -85,B 0,C 180,E1 -4153.932,E2 -4153.932} C_VEL
LIN {X 0,Y 539.295,Z 652.283,A -85,B 0,C 180,E1 -4154.264,E2 -4154.264} C_VEL
LIN {X 0,Y 539.445,Z 618.528,A -85,B 0,C 180,E1 -4154.741,E2 -4154.741} C_VEL
LIN {X 0,Y 539.573,Z 549.388,A -85,B 0,C 180,E1 -4155.668,E2 -4155.668} C_VEL
LIN {X 0,Y 538.428,Z 541.825,A -85,B 0,C 180,E1 -4155.805,E2 -4155.805} C_VEL
LIN {X 0,Y 538.844,Z 521.849,A -85,B 0,C 180,E1 -4158.636,E2 -4158.636} C_VEL
LIN {X 0,Y 539.242,Z 501.179,A -85,B 0,C 180,E1 -4161.604,E2 -4161.604} C_VEL
LIN {X 0,Y 539.681,Z 484.565,A -85,B 0,C 180,E1 -4164.023,E2 -4164.023} C_VEL
LIN {X 0,Y 539.087,Z 482.41,A -85,B 0,C 180,E1 -4164.367,E2 -4164.367} C_VEL
LIN {X 0,Y 536.305,Z 479.462,A -85,B 0,C 180,E1 -4164.933,E2 -4164.933} C_VEL
LIN {X 0,Y 532.743,Z 475.975,A -85,B 0,C 180,E1 -4165.626,E2 -4165.626} C_VEL
LIN {X 0,Y 532.142,Z 474.583,A -85,B 0,C 180,E1 -4165.866,E2 -4165.866} C_VEL
LIN {X 0,Y 531.029,Z 469.464,A -85,B 0,C 180,E1 -4166.715,E2 -4166.715} C_VEL
LIN {X 0,Y 530.985,Z 469.471,A -85,B 0,C 180,E1 -4169.322,E2 -4169.322} C_VEL
LIN {X 0,Y 530.969,Z 469.469,A -85,B 0,C 180,E1 -4172.1,E2 -4172.1} C_VEL
LIN {X 0,Y 530.987,Z 469.464,A -85,B 0,C 180,E1 -4174.853,E2 -4174.853} C_VEL
LIN {X 0,Y 530.969,Z 469.473,A -85,B 0,C 180,E1 -4177.507,E2 -4177.507} C_VEL
LIN {X 0,Y 530.984,Z 469.463,A -85,B 0,C 180,E1 -4180.433,E2 -4180.433} C_VEL
LIN {X 0,Y 530.963,Z 469.47,A -85,B 0,C 180,E1 -4183.281,E2 -4183.281} C_VEL
LIN {X 0,Y 530.985,Z 469.472,A -85,B 0,C 180,E1 -4185.621,E2 -4185.621} C_VEL
LIN {X 0,Y 530.999,Z 469.461,A -85,B 0,C 180,E1 -4188.565,E2 -4188.565} C_VEL
LIN {X 0,Y 530.96,Z 469.475,A -85,B 0,C 180,E1 -4191.529,E2 -4191.529} C_VEL
LIN {X 0,Y 530.956,Z 469.466,A -85,B 0,C 180,E1 -4194.38,E2 -4194.38} C_VEL
LIN {X 0,Y 530.969,Z 469.468,A -85,B 0,C 180,E1 -4197.133,E2 -4197.133} C_VEL
LIN {X 0,Y 530.972,Z 469.47,A -85,B 0,C 180,E1 -4199.803,E2 -4199.803} C_VEL
LIN {X 0,Y 531.015,Z 469.459,A -85,B 0,C 180,E1 -4202.467,E2 -4202.467} C_VEL
LIN {X 0,Y 531.008,Z 469.462,A -85,B 0,C 180,E1 -4204.942,E2 -4204.942} C_VEL
LIN {X 0,Y 530.974,Z 469.465,A -85,B 0,C 180,E1 -4208.247,E2 -4208.247} C_VEL
LIN {X 0,Y 530.998,Z 469.461,A -85,B 0,C 180,E1 -4210.677,E2 -4210.677} C_VEL
